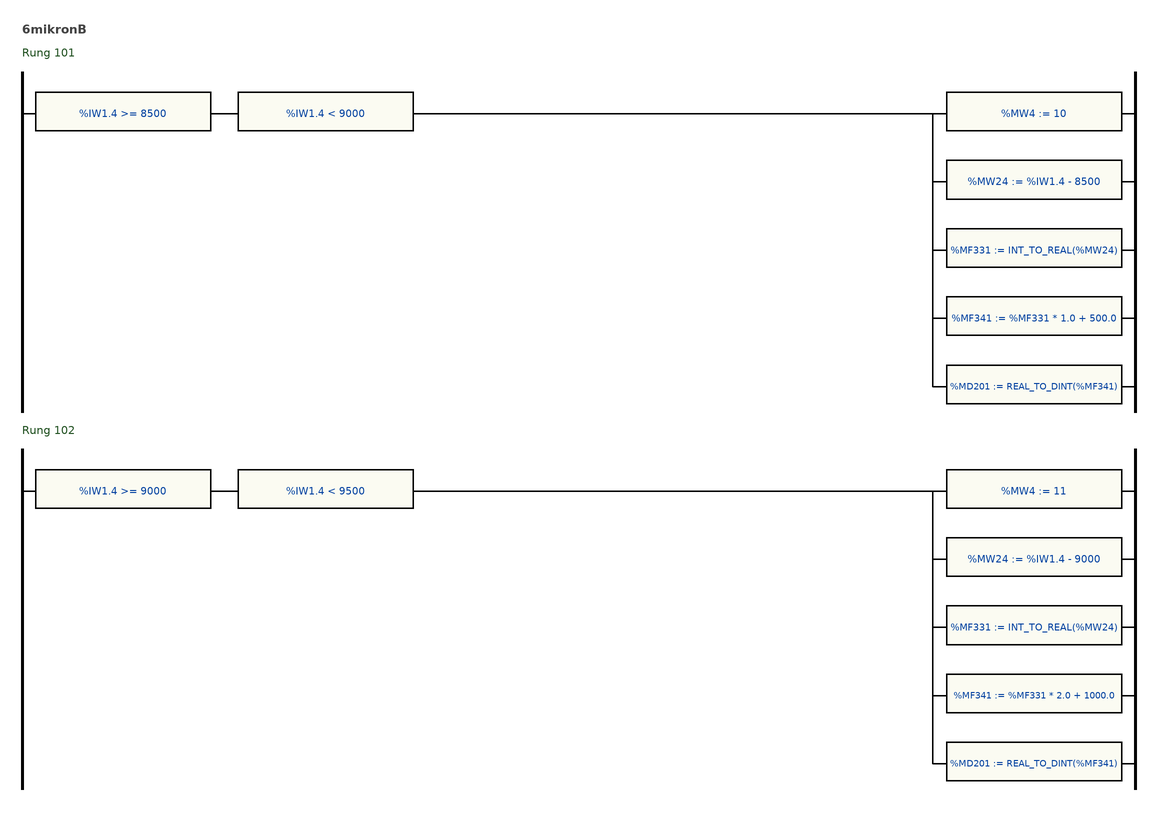
[picture p48: 6mikronB, ladder]

// Rung 101
  LD [ %IW1.4 >= 8500 ]
  AND [ %IW1.4 < 9000 ]
  [ %MW4 := 10 ]
  [ %MW24 := %IW1.4 - 8500 ]
  [ %MF331 := INT_TO_REAL ( %MW24 ) ]
  [ %MF341 := %MF331 * 1.0 + 500.0 ]
  [ %MD201 := REAL_TO_DINT ( %MF341 ) ]
  // as ST:
  //   IF %IW1.4 >= 8500 AND %IW1.4 < 9000 THEN %MW4 := 10; END_IF;
  //   IF %IW1.4 >= 8500 AND %IW1.4 < 9000 THEN %MW24 := %IW1.4 - 8500; END_IF;
  //   IF %IW1.4 >= 8500 AND %IW1.4 < 9000 THEN %MF331 := INT_TO_REAL ( %MW24 ); END_IF;
  //   IF %IW1.4 >= 8500 AND %IW1.4 < 9000 THEN %MF341 := %MF331 * 1.0 + 500.0; END_IF;
  //   IF %IW1.4 >= 8500 AND %IW1.4 < 9000 THEN %MD201 := REAL_TO_DINT ( %MF341 ); END_IF;

// Rung 102
  LD [ %IW1.4 >= 9000 ]
  AND [ %IW1.4 < 9500 ]
  [ %MW4 := 11 ]
  [ %MW24 := %IW1.4 - 9000 ]
  [ %MF331 := INT_TO_REAL ( %MW24 ) ]
  [ %MF341 := %MF331 * 2.0 + 1000.0 ]
  [ %MD201 := REAL_TO_DINT ( %MF341 ) ]
  // as ST:
  //   IF %IW1.4 >= 9000 AND %IW1.4 < 9500 THEN %MW4 := 11; END_IF;
  //   IF %IW1.4 >= 9000 AND %IW1.4 < 9500 THEN %MW24 := %IW1.4 - 9000; END_IF;
  //   IF %IW1.4 >= 9000 AND %IW1.4 < 9500 THEN %MF331 := INT_TO_REAL ( %MW24 ); END_IF;
  //   IF %IW1.4 >= 9000 AND %IW1.4 < 9500 THEN %MF341 := %MF331 * 2.0 + 1000.0; END_IF;
  //   IF %IW1.4 >= 9000 AND %IW1.4 < 9500 THEN %MD201 := REAL_TO_DINT ( %MF341 ); END_IF;

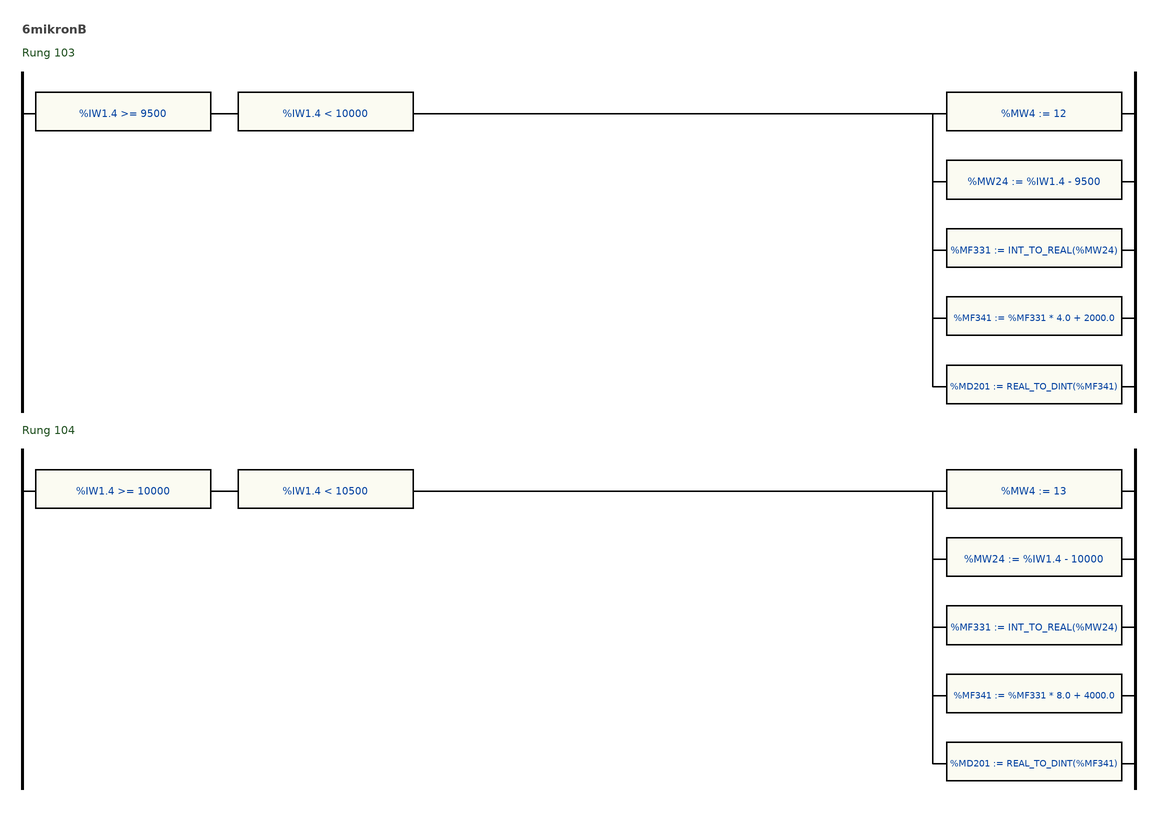

// Rung 103
  LD [ %IW1.4 >= 9500 ]
  AND [ %IW1.4 < 10000 ]
  [ %MW4 := 12 ]
  [ %MW24 := %IW1.4 - 9500 ]
  [ %MF331 := INT_TO_REAL ( %MW24 ) ]
  [ %MF341 := %MF331 * 4.0 + 2000.0 ]
  [ %MD201 := REAL_TO_DINT ( %MF341 ) ]
  // as ST:
  //   IF %IW1.4 >= 9500 AND %IW1.4 < 10000 THEN %MW4 := 12; END_IF;
  //   IF %IW1.4 >= 9500 AND %IW1.4 < 10000 THEN %MW24 := %IW1.4 - 9500; END_IF;
  //   IF %IW1.4 >= 9500 AND %IW1.4 < 10000 THEN %MF331 := INT_TO_REAL ( %MW24 ); END_IF;
  //   IF %IW1.4 >= 9500 AND %IW1.4 < 10000 THEN %MF341 := %MF331 * 4.0 + 2000.0; END_IF;
  //   IF %IW1.4 >= 9500 AND %IW1.4 < 10000 THEN %MD201 := REAL_TO_DINT ( %MF341 ); END_IF;

// Rung 104
  LD [ %IW1.4 >= 10000 ]
  AND [ %IW1.4 < 10500 ]
  [ %MW4 := 13 ]
  [ %MW24 := %IW1.4 - 10000 ]
  [ %MF331 := INT_TO_REAL ( %MW24 ) ]
  [ %MF341 := %MF331 * 8.0 + 4000.0 ]
  [ %MD201 := REAL_TO_DINT ( %MF341 ) ]
  // as ST:
  //   IF %IW1.4 >= 10000 AND %IW1.4 < 10500 THEN %MW4 := 13; END_IF;
  //   IF %IW1.4 >= 10000 AND %IW1.4 < 10500 THEN %MW24 := %IW1.4 - 10000; END_IF;
  //   IF %IW1.4 >= 10000 AND %IW1.4 < 10500 THEN %MF331 := INT_TO_REAL ( %MW24 ); END_IF;
  //   IF %IW1.4 >= 10000 AND %IW1.4 < 10500 THEN %MF341 := %MF331 * 8.0 + 4000.0; END_IF;
  //   IF %IW1.4 >= 10000 AND %IW1.4 < 10500 THEN %MD201 := REAL_TO_DINT ( %MF341 ); END_IF;

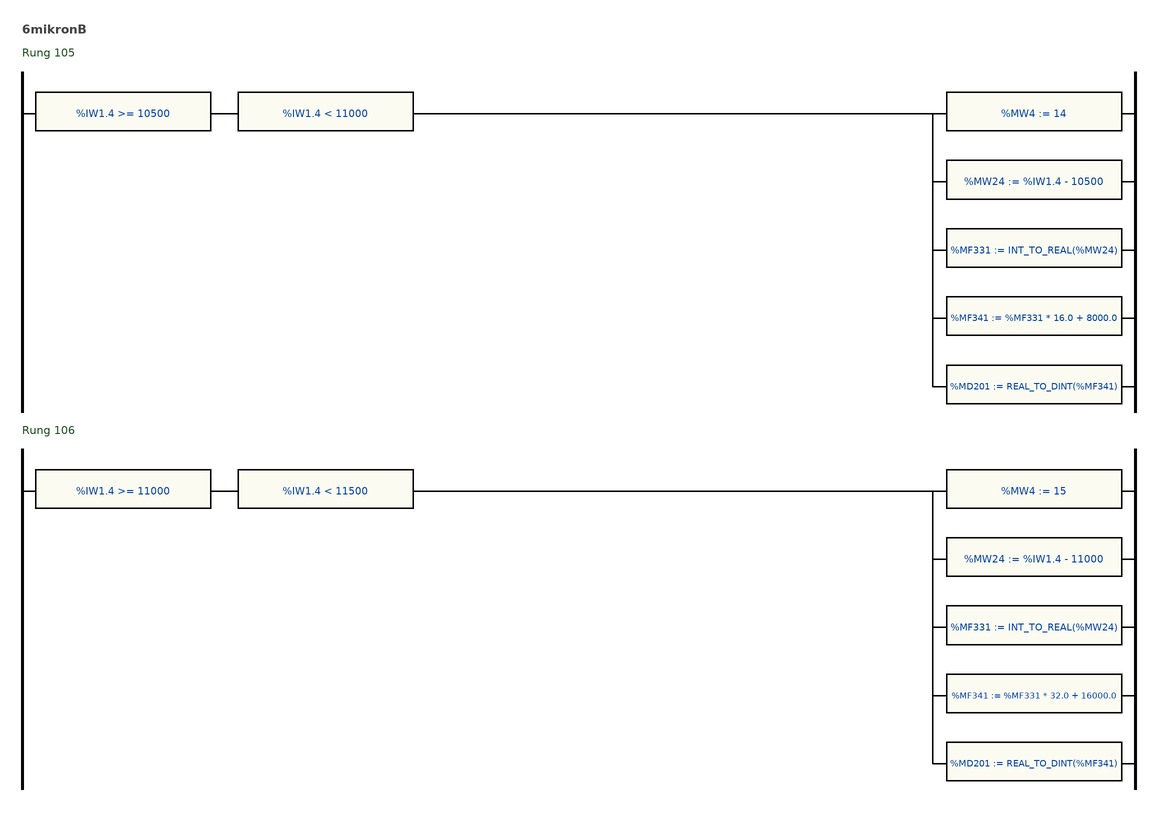

// Rung 105
  LD [ %IW1.4 >= 10500 ]
  AND [ %IW1.4 < 11000 ]
  [ %MW4 := 14 ]
  [ %MW24 := %IW1.4 - 10500 ]
  [ %MF331 := INT_TO_REAL ( %MW24 ) ]
  [ %MF341 := %MF331 * 16.0 + 8000.0 ]
  [ %MD201 := REAL_TO_DINT ( %MF341 ) ]
  // as ST:
  //   IF %IW1.4 >= 10500 AND %IW1.4 < 11000 THEN %MW4 := 14; END_IF;
  //   IF %IW1.4 >= 10500 AND %IW1.4 < 11000 THEN %MW24 := %IW1.4 - 10500; END_IF;
  //   IF %IW1.4 >= 10500 AND %IW1.4 < 11000 THEN %MF331 := INT_TO_REAL ( %MW24 ); END_IF;
  //   IF %IW1.4 >= 10500 AND %IW1.4 < 11000 THEN %MF341 := %MF331 * 16.0 + 8000.0; END_IF;
  //   IF %IW1.4 >= 10500 AND %IW1.4 < 11000 THEN %MD201 := REAL_TO_DINT ( %MF341 ); END_IF;

// Rung 106
  LD [ %IW1.4 >= 11000 ]
  AND [ %IW1.4 < 11500 ]
  [ %MW4 := 15 ]
  [ %MW24 := %IW1.4 - 11000 ]
  [ %MF331 := INT_TO_REAL ( %MW24 ) ]
  [ %MF341 := %MF331 * 32.0 + 16000.0 ]
  [ %MD201 := REAL_TO_DINT ( %MF341 ) ]
  // as ST:
  //   IF %IW1.4 >= 11000 AND %IW1.4 < 11500 THEN %MW4 := 15; END_IF;
  //   IF %IW1.4 >= 11000 AND %IW1.4 < 11500 THEN %MW24 := %IW1.4 - 11000; END_IF;
  //   IF %IW1.4 >= 11000 AND %IW1.4 < 11500 THEN %MF331 := INT_TO_REAL ( %MW24 ); END_IF;
  //   IF %IW1.4 >= 11000 AND %IW1.4 < 11500 THEN %MF341 := %MF331 * 32.0 + 16000.0; END_IF;
  //   IF %IW1.4 >= 11000 AND %IW1.4 < 11500 THEN %MD201 := REAL_TO_DINT ( %MF341 ); END_IF;

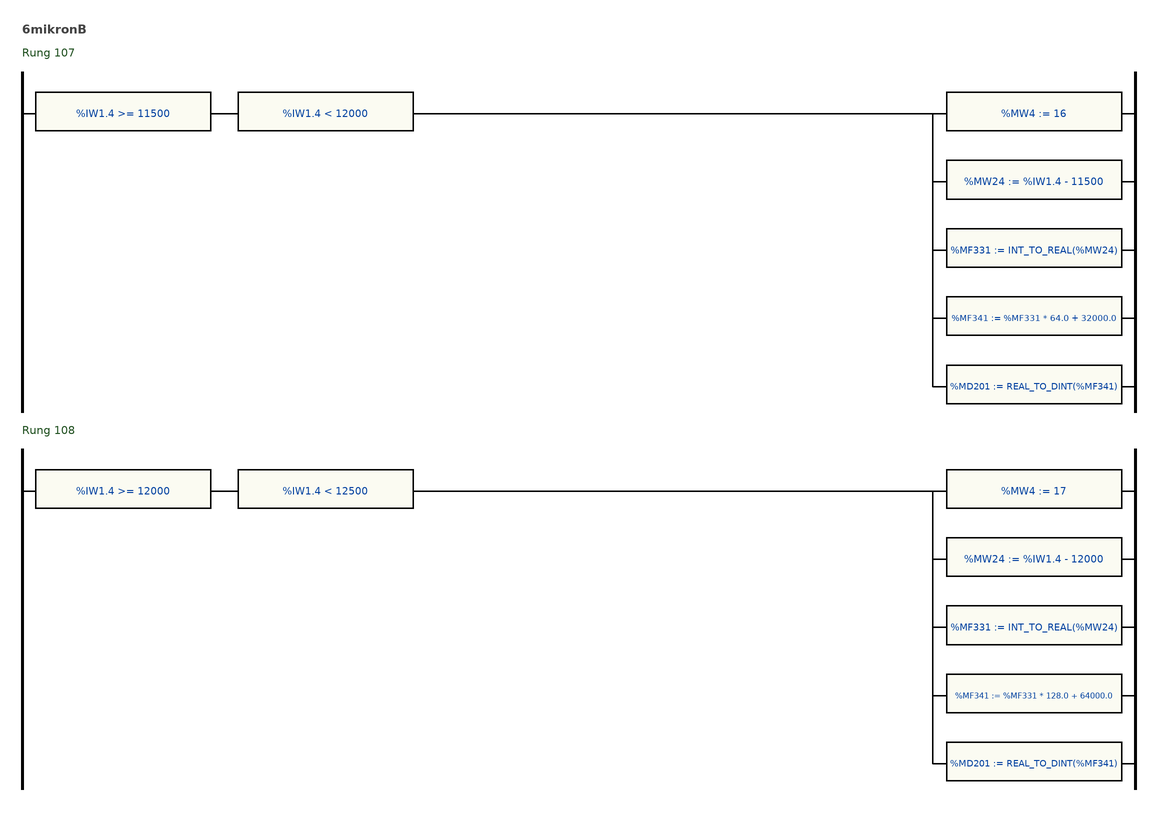

// Rung 107
  LD [ %IW1.4 >= 11500 ]
  AND [ %IW1.4 < 12000 ]
  [ %MW4 := 16 ]
  [ %MW24 := %IW1.4 - 11500 ]
  [ %MF331 := INT_TO_REAL ( %MW24 ) ]
  [ %MF341 := %MF331 * 64.0 + 32000.0 ]
  [ %MD201 := REAL_TO_DINT ( %MF341 ) ]
  // as ST:
  //   IF %IW1.4 >= 11500 AND %IW1.4 < 12000 THEN %MW4 := 16; END_IF;
  //   IF %IW1.4 >= 11500 AND %IW1.4 < 12000 THEN %MW24 := %IW1.4 - 11500; END_IF;
  //   IF %IW1.4 >= 11500 AND %IW1.4 < 12000 THEN %MF331 := INT_TO_REAL ( %MW24 ); END_IF;
  //   IF %IW1.4 >= 11500 AND %IW1.4 < 12000 THEN %MF341 := %MF331 * 64.0 + 32000.0; END_IF;
  //   IF %IW1.4 >= 11500 AND %IW1.4 < 12000 THEN %MD201 := REAL_TO_DINT ( %MF341 ); END_IF;

// Rung 108
  LD [ %IW1.4 >= 12000 ]
  AND [ %IW1.4 < 12500 ]
  [ %MW4 := 17 ]
  [ %MW24 := %IW1.4 - 12000 ]
  [ %MF331 := INT_TO_REAL ( %MW24 ) ]
  [ %MF341 := %MF331 * 128.0 + 64000.0 ]
  [ %MD201 := REAL_TO_DINT ( %MF341 ) ]
  // as ST:
  //   IF %IW1.4 >= 12000 AND %IW1.4 < 12500 THEN %MW4 := 17; END_IF;
  //   IF %IW1.4 >= 12000 AND %IW1.4 < 12500 THEN %MW24 := %IW1.4 - 12000; END_IF;
  //   IF %IW1.4 >= 12000 AND %IW1.4 < 12500 THEN %MF331 := INT_TO_REAL ( %MW24 ); END_IF;
  //   IF %IW1.4 >= 12000 AND %IW1.4 < 12500 THEN %MF341 := %MF331 * 128.0 + 64000.0; END_IF;
  //   IF %IW1.4 >= 12000 AND %IW1.4 < 12500 THEN %MD201 := REAL_TO_DINT ( %MF341 ); END_IF;

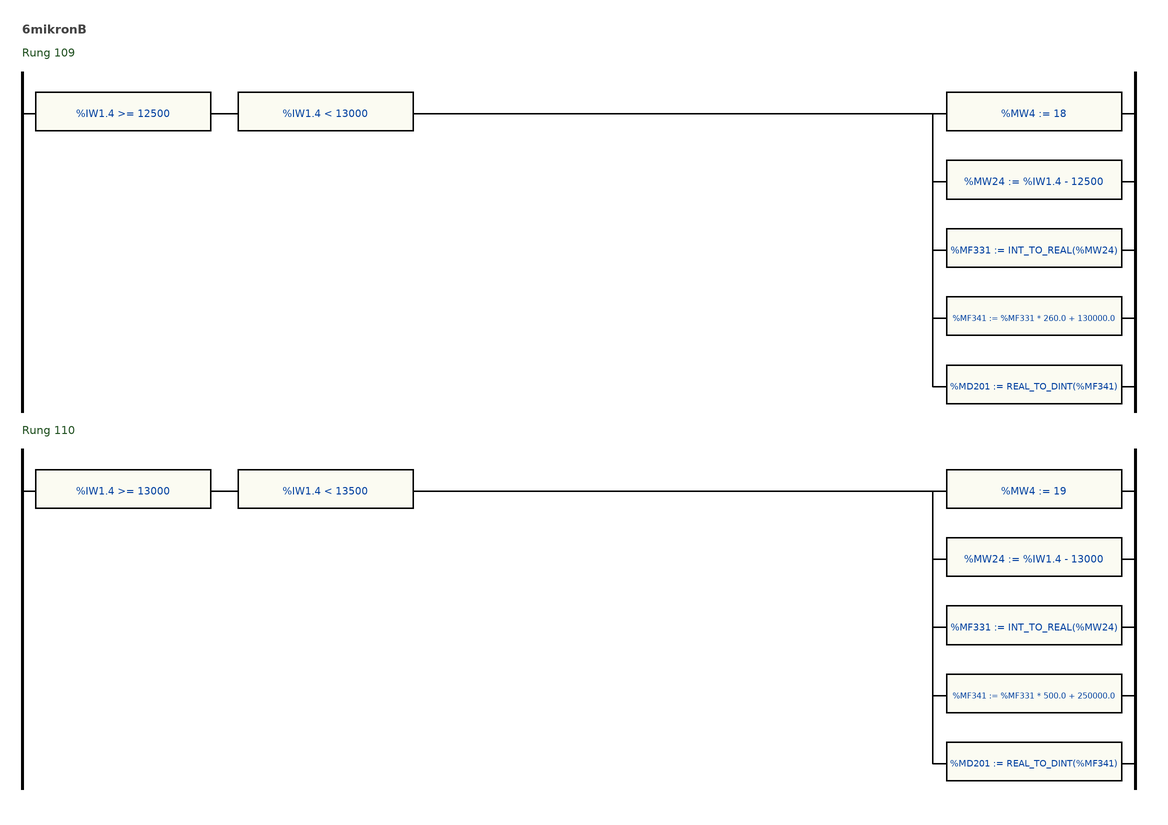

// Rung 109
  LD [ %IW1.4 >= 12500 ]
  AND [ %IW1.4 < 13000 ]
  [ %MW4 := 18 ]
  [ %MW24 := %IW1.4 - 12500 ]
  [ %MF331 := INT_TO_REAL ( %MW24 ) ]
  [ %MF341 := %MF331 * 260.0 + 130000.0 ]
  [ %MD201 := REAL_TO_DINT ( %MF341 ) ]
  // as ST:
  //   IF %IW1.4 >= 12500 AND %IW1.4 < 13000 THEN %MW4 := 18; END_IF;
  //   IF %IW1.4 >= 12500 AND %IW1.4 < 13000 THEN %MW24 := %IW1.4 - 12500; END_IF;
  //   IF %IW1.4 >= 12500 AND %IW1.4 < 13000 THEN %MF331 := INT_TO_REAL ( %MW24 ); END_IF;
  //   IF %IW1.4 >= 12500 AND %IW1.4 < 13000 THEN %MF341 := %MF331 * 260.0 + 130000.0; END_IF;
  //   IF %IW1.4 >= 12500 AND %IW1.4 < 13000 THEN %MD201 := REAL_TO_DINT ( %MF341 ); END_IF;

// Rung 110
  LD [ %IW1.4 >= 13000 ]
  AND [ %IW1.4 < 13500 ]
  [ %MW4 := 19 ]
  [ %MW24 := %IW1.4 - 13000 ]
  [ %MF331 := INT_TO_REAL ( %MW24 ) ]
  [ %MF341 := %MF331 * 500.0 + 250000.0 ]
  [ %MD201 := REAL_TO_DINT ( %MF341 ) ]
  // as ST:
  //   IF %IW1.4 >= 13000 AND %IW1.4 < 13500 THEN %MW4 := 19; END_IF;
  //   IF %IW1.4 >= 13000 AND %IW1.4 < 13500 THEN %MW24 := %IW1.4 - 13000; END_IF;
  //   IF %IW1.4 >= 13000 AND %IW1.4 < 13500 THEN %MF331 := INT_TO_REAL ( %MW24 ); END_IF;
  //   IF %IW1.4 >= 13000 AND %IW1.4 < 13500 THEN %MF341 := %MF331 * 500.0 + 250000.0; END_IF;
  //   IF %IW1.4 >= 13000 AND %IW1.4 < 13500 THEN %MD201 := REAL_TO_DINT ( %MF341 ); END_IF;

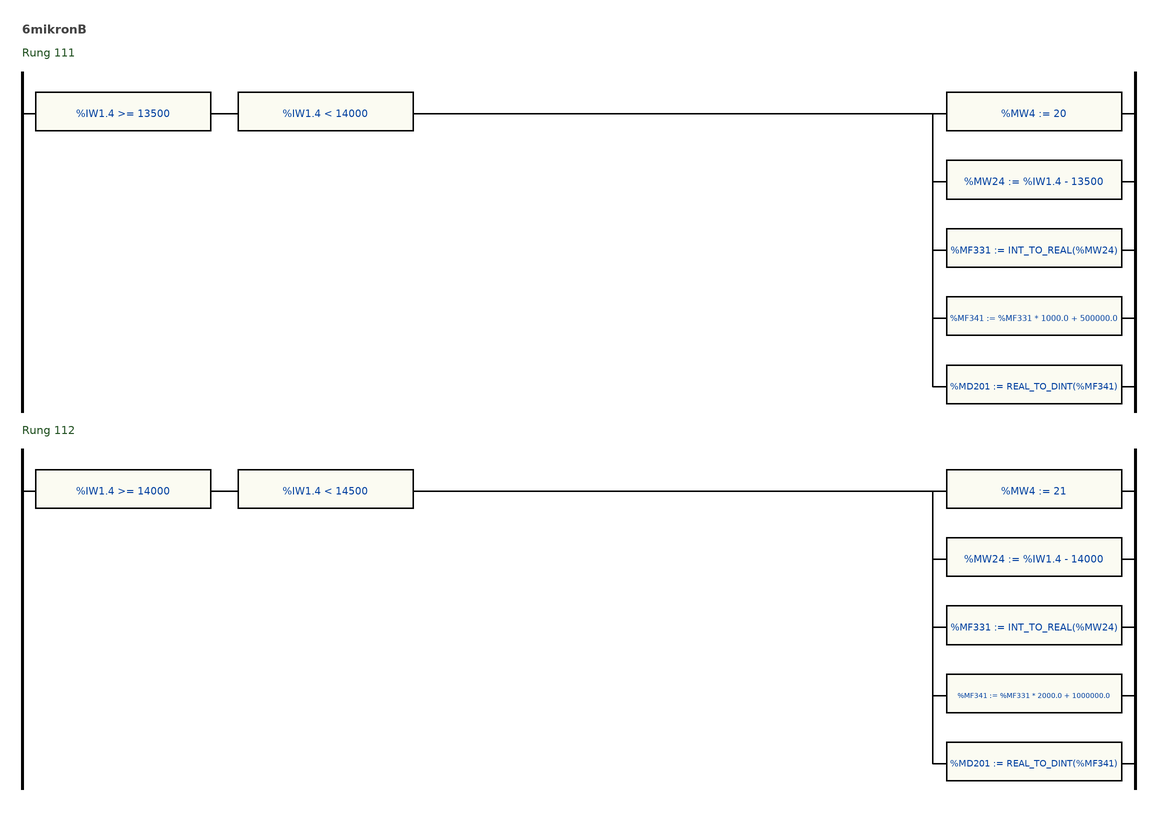

// Rung 111
  LD [ %IW1.4 >= 13500 ]
  AND [ %IW1.4 < 14000 ]
  [ %MW4 := 20 ]
  [ %MW24 := %IW1.4 - 13500 ]
  [ %MF331 := INT_TO_REAL ( %MW24 ) ]
  [ %MF341 := %MF331 * 1000.0 + 500000.0 ]
  [ %MD201 := REAL_TO_DINT ( %MF341 ) ]
  // as ST:
  //   IF %IW1.4 >= 13500 AND %IW1.4 < 14000 THEN %MW4 := 20; END_IF;
  //   IF %IW1.4 >= 13500 AND %IW1.4 < 14000 THEN %MW24 := %IW1.4 - 13500; END_IF;
  //   IF %IW1.4 >= 13500 AND %IW1.4 < 14000 THEN %MF331 := INT_TO_REAL ( %MW24 ); END_IF;
  //   IF %IW1.4 >= 13500 AND %IW1.4 < 14000 THEN %MF341 := %MF331 * 1000.0 + 500000.0; END_IF;
  //   IF %IW1.4 >= 13500 AND %IW1.4 < 14000 THEN %MD201 := REAL_TO_DINT ( %MF341 ); END_IF;

// Rung 112
  LD [ %IW1.4 >= 14000 ]
  AND [ %IW1.4 < 14500 ]
  [ %MW4 := 21 ]
  [ %MW24 := %IW1.4 - 14000 ]
  [ %MF331 := INT_TO_REAL ( %MW24 ) ]
  [ %MF341 := %MF331 * 2000.0 + 1000000.0 ]
  [ %MD201 := REAL_TO_DINT ( %MF341 ) ]
  // as ST:
  //   IF %IW1.4 >= 14000 AND %IW1.4 < 14500 THEN %MW4 := 21; END_IF;
  //   IF %IW1.4 >= 14000 AND %IW1.4 < 14500 THEN %MW24 := %IW1.4 - 14000; END_IF;
  //   IF %IW1.4 >= 14000 AND %IW1.4 < 14500 THEN %MF331 := INT_TO_REAL ( %MW24 ); END_IF;
  //   IF %IW1.4 >= 14000 AND %IW1.4 < 14500 THEN %MF341 := %MF331 * 2000.0 + 1000000.0; END_IF;
  //   IF %IW1.4 >= 14000 AND %IW1.4 < 14500 THEN %MD201 := REAL_TO_DINT ( %MF341 ); END_IF;

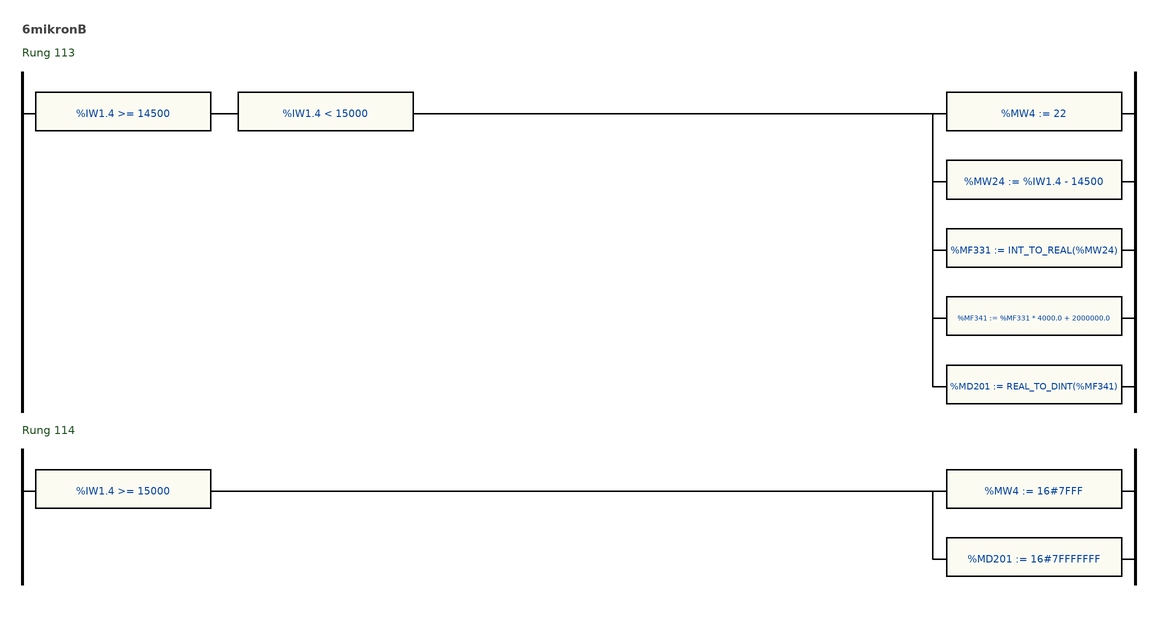

// Rung 113
  LD [ %IW1.4 >= 14500 ]
  AND [ %IW1.4 < 15000 ]
  [ %MW4 := 22 ]
  [ %MW24 := %IW1.4 - 14500 ]
  [ %MF331 := INT_TO_REAL ( %MW24 ) ]
  [ %MF341 := %MF331 * 4000.0 + 2000000.0 ]
  [ %MD201 := REAL_TO_DINT ( %MF341 ) ]
  // as ST:
  //   IF %IW1.4 >= 14500 AND %IW1.4 < 15000 THEN %MW4 := 22; END_IF;
  //   IF %IW1.4 >= 14500 AND %IW1.4 < 15000 THEN %MW24 := %IW1.4 - 14500; END_IF;
  //   IF %IW1.4 >= 14500 AND %IW1.4 < 15000 THEN %MF331 := INT_TO_REAL ( %MW24 ); END_IF;
  //   IF %IW1.4 >= 14500 AND %IW1.4 < 15000 THEN %MF341 := %MF331 * 4000.0 + 2000000.0; END_IF;
  //   IF %IW1.4 >= 14500 AND %IW1.4 < 15000 THEN %MD201 := REAL_TO_DINT ( %MF341 ); END_IF;

// Rung 114
  LD [ %IW1.4 >= 15000 ]
  [ %MW4 := 16#7FFF ]
  [ %MD201 := 16#7FFFFFFF ]
  // as ST:
  //   IF %IW1.4 >= 15000 THEN %MW4 := 16#7FFF; END_IF;
  //   IF %IW1.4 >= 15000 THEN %MD201 := 16#7FFFFFFF; END_IF;

POU 14mikronB
  (* SectionNumber=6 *)

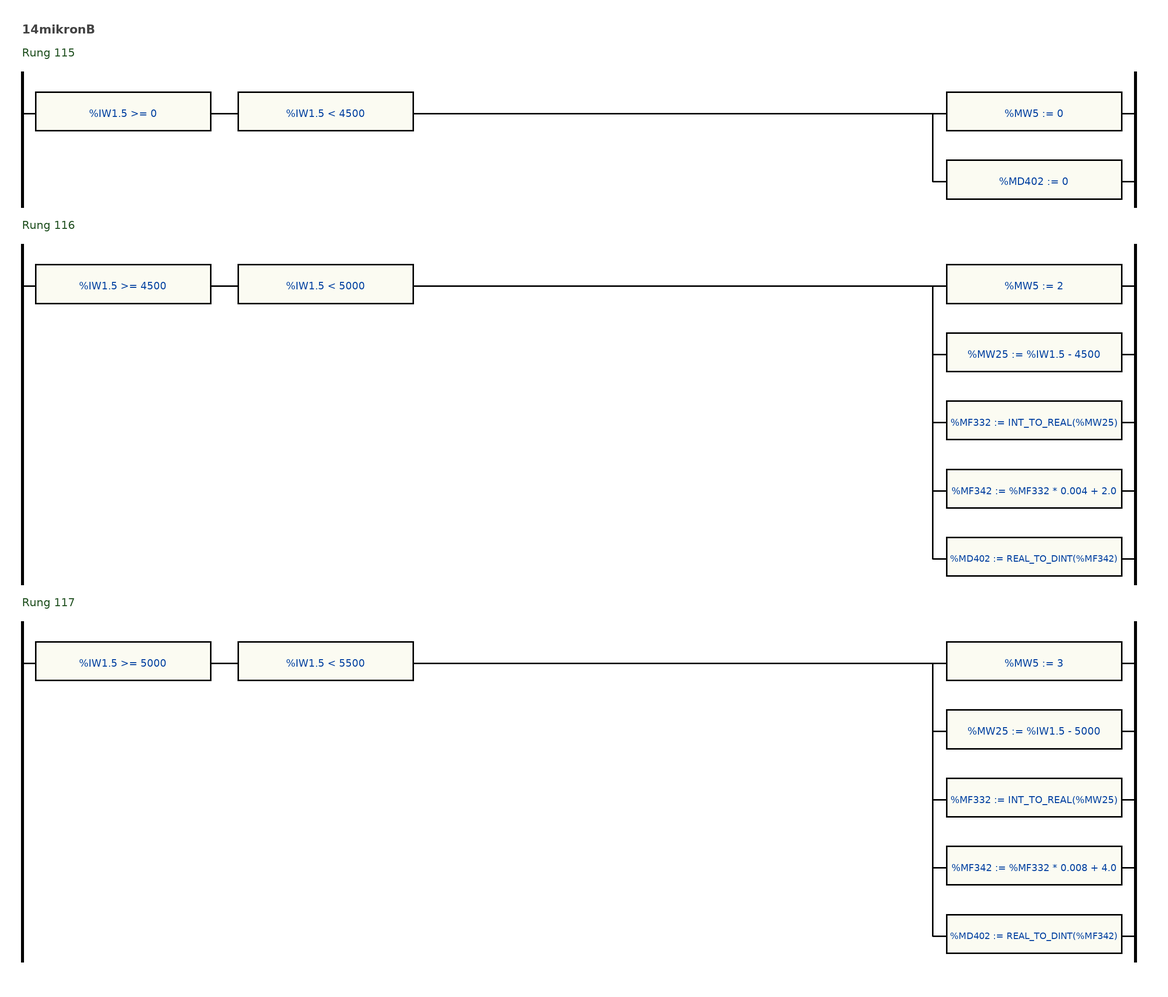

// Rung 115
  LD [ %IW1.5 >= 0 ]
  AND [ %IW1.5 < 4500 ]
  [ %MW5 := 0 ]
  [ %MD402 := 0 ]
  // as ST:
  //   IF %IW1.5 >= 0 AND %IW1.5 < 4500 THEN %MW5 := 0; END_IF;
  //   IF %IW1.5 >= 0 AND %IW1.5 < 4500 THEN %MD402 := 0; END_IF;

// Rung 116
  LD [ %IW1.5 >= 4500 ]
  AND [ %IW1.5 < 5000 ]
  [ %MW5 := 2 ]
  [ %MW25 := %IW1.5 - 4500 ]
  [ %MF332 := INT_TO_REAL ( %MW25 ) ]
  [ %MF342 := %MF332 * 0.004 + 2.0 ]
  [ %MD402 := REAL_TO_DINT ( %MF342 ) ]
  // as ST:
  //   IF %IW1.5 >= 4500 AND %IW1.5 < 5000 THEN %MW5 := 2; END_IF;
  //   IF %IW1.5 >= 4500 AND %IW1.5 < 5000 THEN %MW25 := %IW1.5 - 4500; END_IF;
  //   IF %IW1.5 >= 4500 AND %IW1.5 < 5000 THEN %MF332 := INT_TO_REAL ( %MW25 ); END_IF;
  //   IF %IW1.5 >= 4500 AND %IW1.5 < 5000 THEN %MF342 := %MF332 * 0.004 + 2.0; END_IF;
  //   IF %IW1.5 >= 4500 AND %IW1.5 < 5000 THEN %MD402 := REAL_TO_DINT ( %MF342 ); END_IF;

// Rung 117
  LD [ %IW1.5 >= 5000 ]
  AND [ %IW1.5 < 5500 ]
  [ %MW5 := 3 ]
  [ %MW25 := %IW1.5 - 5000 ]
  [ %MF332 := INT_TO_REAL ( %MW25 ) ]
  [ %MF342 := %MF332 * 0.008 + 4.0 ]
  [ %MD402 := REAL_TO_DINT ( %MF342 ) ]
  // as ST:
  //   IF %IW1.5 >= 5000 AND %IW1.5 < 5500 THEN %MW5 := 3; END_IF;
  //   IF %IW1.5 >= 5000 AND %IW1.5 < 5500 THEN %MW25 := %IW1.5 - 5000; END_IF;
  //   IF %IW1.5 >= 5000 AND %IW1.5 < 5500 THEN %MF332 := INT_TO_REAL ( %MW25 ); END_IF;
  //   IF %IW1.5 >= 5000 AND %IW1.5 < 5500 THEN %MF342 := %MF332 * 0.008 + 4.0; END_IF;
  //   IF %IW1.5 >= 5000 AND %IW1.5 < 5500 THEN %MD402 := REAL_TO_DINT ( %MF342 ); END_IF;

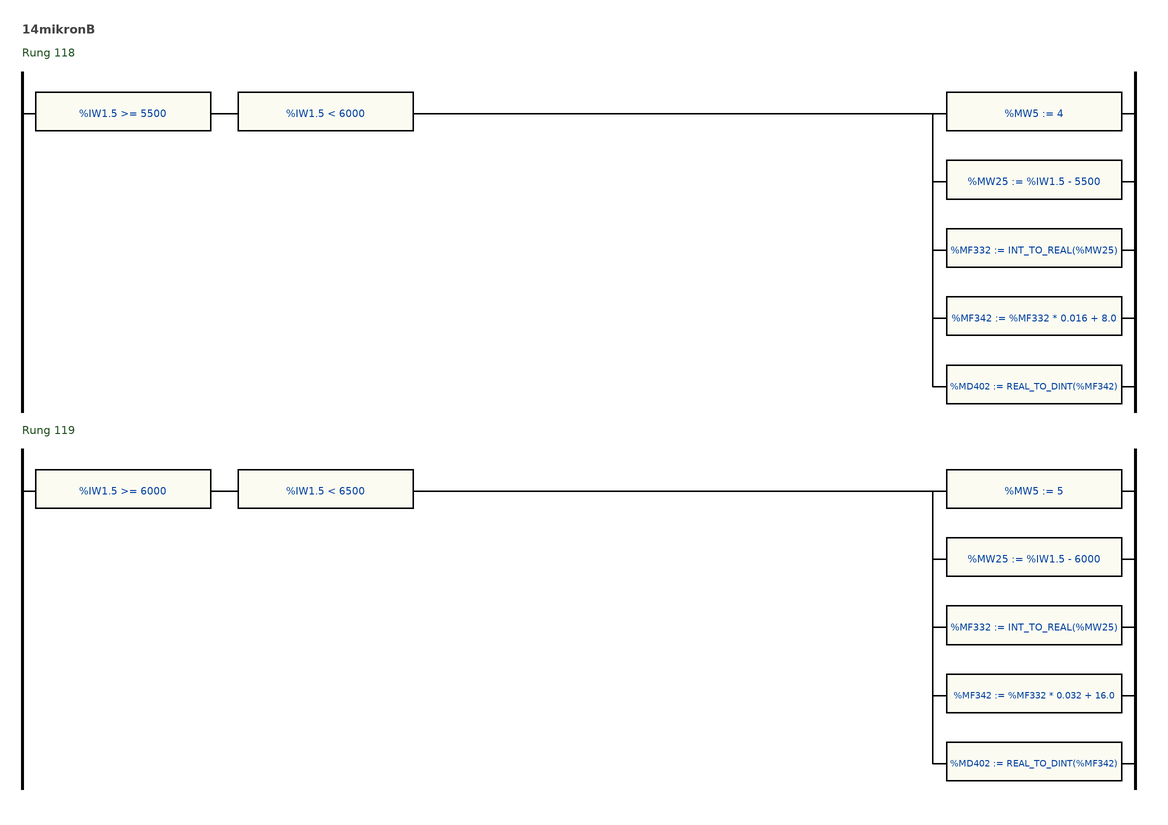

// Rung 118
  LD [ %IW1.5 >= 5500 ]
  AND [ %IW1.5 < 6000 ]
  [ %MW5 := 4 ]
  [ %MW25 := %IW1.5 - 5500 ]
  [ %MF332 := INT_TO_REAL ( %MW25 ) ]
  [ %MF342 := %MF332 * 0.016 + 8.0 ]
  [ %MD402 := REAL_TO_DINT ( %MF342 ) ]
  // as ST:
  //   IF %IW1.5 >= 5500 AND %IW1.5 < 6000 THEN %MW5 := 4; END_IF;
  //   IF %IW1.5 >= 5500 AND %IW1.5 < 6000 THEN %MW25 := %IW1.5 - 5500; END_IF;
  //   IF %IW1.5 >= 5500 AND %IW1.5 < 6000 THEN %MF332 := INT_TO_REAL ( %MW25 ); END_IF;
  //   IF %IW1.5 >= 5500 AND %IW1.5 < 6000 THEN %MF342 := %MF332 * 0.016 + 8.0; END_IF;
  //   IF %IW1.5 >= 5500 AND %IW1.5 < 6000 THEN %MD402 := REAL_TO_DINT ( %MF342 ); END_IF;

// Rung 119
  LD [ %IW1.5 >= 6000 ]
  AND [ %IW1.5 < 6500 ]
  [ %MW5 := 5 ]
  [ %MW25 := %IW1.5 - 6000 ]
  [ %MF332 := INT_TO_REAL ( %MW25 ) ]
  [ %MF342 := %MF332 * 0.032 + 16.0 ]
  [ %MD402 := REAL_TO_DINT ( %MF342 ) ]
  // as ST:
  //   IF %IW1.5 >= 6000 AND %IW1.5 < 6500 THEN %MW5 := 5; END_IF;
  //   IF %IW1.5 >= 6000 AND %IW1.5 < 6500 THEN %MW25 := %IW1.5 - 6000; END_IF;
  //   IF %IW1.5 >= 6000 AND %IW1.5 < 6500 THEN %MF332 := INT_TO_REAL ( %MW25 ); END_IF;
  //   IF %IW1.5 >= 6000 AND %IW1.5 < 6500 THEN %MF342 := %MF332 * 0.032 + 16.0; END_IF;
  //   IF %IW1.5 >= 6000 AND %IW1.5 < 6500 THEN %MD402 := REAL_TO_DINT ( %MF342 ); END_IF;

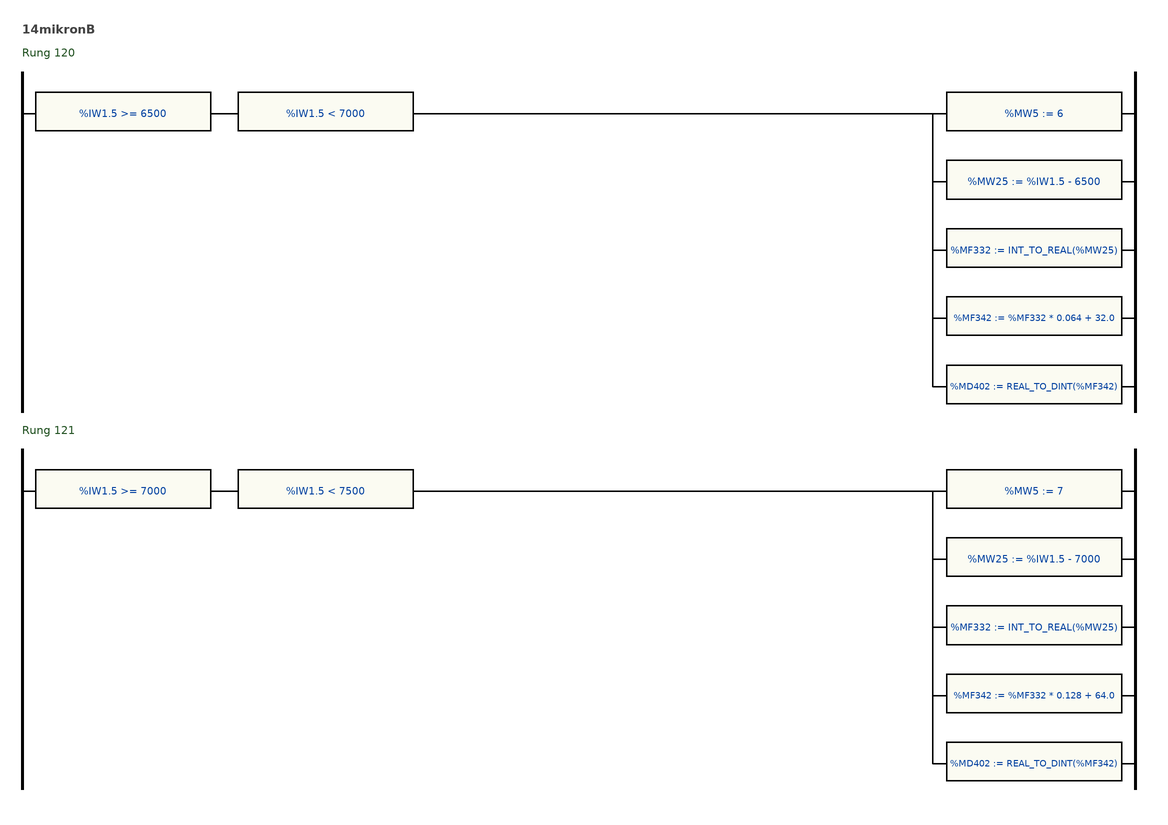

// Rung 120
  LD [ %IW1.5 >= 6500 ]
  AND [ %IW1.5 < 7000 ]
  [ %MW5 := 6 ]
  [ %MW25 := %IW1.5 - 6500 ]
  [ %MF332 := INT_TO_REAL ( %MW25 ) ]
  [ %MF342 := %MF332 * 0.064 + 32.0 ]
  [ %MD402 := REAL_TO_DINT ( %MF342 ) ]
  // as ST:
  //   IF %IW1.5 >= 6500 AND %IW1.5 < 7000 THEN %MW5 := 6; END_IF;
  //   IF %IW1.5 >= 6500 AND %IW1.5 < 7000 THEN %MW25 := %IW1.5 - 6500; END_IF;
  //   IF %IW1.5 >= 6500 AND %IW1.5 < 7000 THEN %MF332 := INT_TO_REAL ( %MW25 ); END_IF;
  //   IF %IW1.5 >= 6500 AND %IW1.5 < 7000 THEN %MF342 := %MF332 * 0.064 + 32.0; END_IF;
  //   IF %IW1.5 >= 6500 AND %IW1.5 < 7000 THEN %MD402 := REAL_TO_DINT ( %MF342 ); END_IF;

// Rung 121
  LD [ %IW1.5 >= 7000 ]
  AND [ %IW1.5 < 7500 ]
  [ %MW5 := 7 ]
  [ %MW25 := %IW1.5 - 7000 ]
  [ %MF332 := INT_TO_REAL ( %MW25 ) ]
  [ %MF342 := %MF332 * 0.128 + 64.0 ]
  [ %MD402 := REAL_TO_DINT ( %MF342 ) ]
  // as ST:
  //   IF %IW1.5 >= 7000 AND %IW1.5 < 7500 THEN %MW5 := 7; END_IF;
  //   IF %IW1.5 >= 7000 AND %IW1.5 < 7500 THEN %MW25 := %IW1.5 - 7000; END_IF;
  //   IF %IW1.5 >= 7000 AND %IW1.5 < 7500 THEN %MF332 := INT_TO_REAL ( %MW25 ); END_IF;
  //   IF %IW1.5 >= 7000 AND %IW1.5 < 7500 THEN %MF342 := %MF332 * 0.128 + 64.0; END_IF;
  //   IF %IW1.5 >= 7000 AND %IW1.5 < 7500 THEN %MD402 := REAL_TO_DINT ( %MF342 ); END_IF;

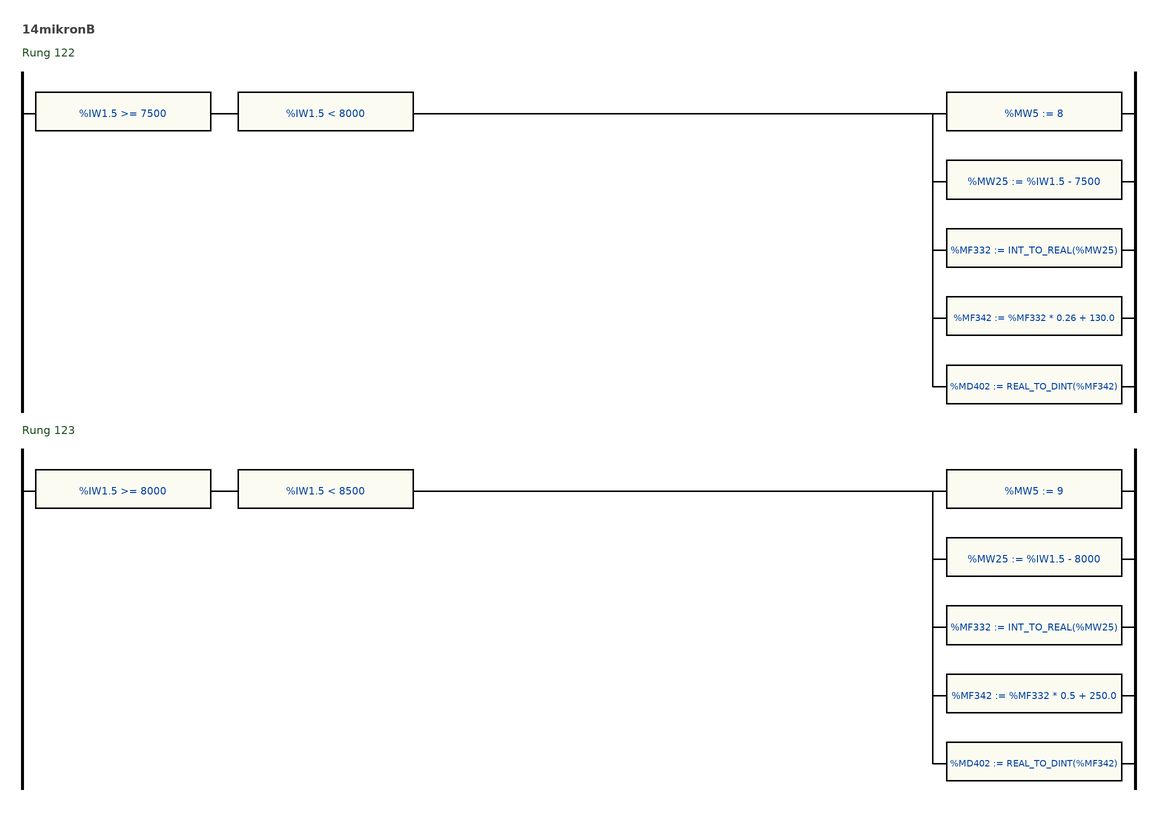

// Rung 122
  LD [ %IW1.5 >= 7500 ]
  AND [ %IW1.5 < 8000 ]
  [ %MW5 := 8 ]
  [ %MW25 := %IW1.5 - 7500 ]
  [ %MF332 := INT_TO_REAL ( %MW25 ) ]
  [ %MF342 := %MF332 * 0.26 + 130.0 ]
  [ %MD402 := REAL_TO_DINT ( %MF342 ) ]
  // as ST:
  //   IF %IW1.5 >= 7500 AND %IW1.5 < 8000 THEN %MW5 := 8; END_IF;
  //   IF %IW1.5 >= 7500 AND %IW1.5 < 8000 THEN %MW25 := %IW1.5 - 7500; END_IF;
  //   IF %IW1.5 >= 7500 AND %IW1.5 < 8000 THEN %MF332 := INT_TO_REAL ( %MW25 ); END_IF;
  //   IF %IW1.5 >= 7500 AND %IW1.5 < 8000 THEN %MF342 := %MF332 * 0.26 + 130.0; END_IF;
  //   IF %IW1.5 >= 7500 AND %IW1.5 < 8000 THEN %MD402 := REAL_TO_DINT ( %MF342 ); END_IF;

// Rung 123
  LD [ %IW1.5 >= 8000 ]
  AND [ %IW1.5 < 8500 ]
  [ %MW5 := 9 ]
  [ %MW25 := %IW1.5 - 8000 ]
  [ %MF332 := INT_TO_REAL ( %MW25 ) ]
  [ %MF342 := %MF332 * 0.5 + 250.0 ]
  [ %MD402 := REAL_TO_DINT ( %MF342 ) ]
  // as ST:
  //   IF %IW1.5 >= 8000 AND %IW1.5 < 8500 THEN %MW5 := 9; END_IF;
  //   IF %IW1.5 >= 8000 AND %IW1.5 < 8500 THEN %MW25 := %IW1.5 - 8000; END_IF;
  //   IF %IW1.5 >= 8000 AND %IW1.5 < 8500 THEN %MF332 := INT_TO_REAL ( %MW25 ); END_IF;
  //   IF %IW1.5 >= 8000 AND %IW1.5 < 8500 THEN %MF342 := %MF332 * 0.5 + 250.0; END_IF;
  //   IF %IW1.5 >= 8000 AND %IW1.5 < 8500 THEN %MD402 := REAL_TO_DINT ( %MF342 ); END_IF;

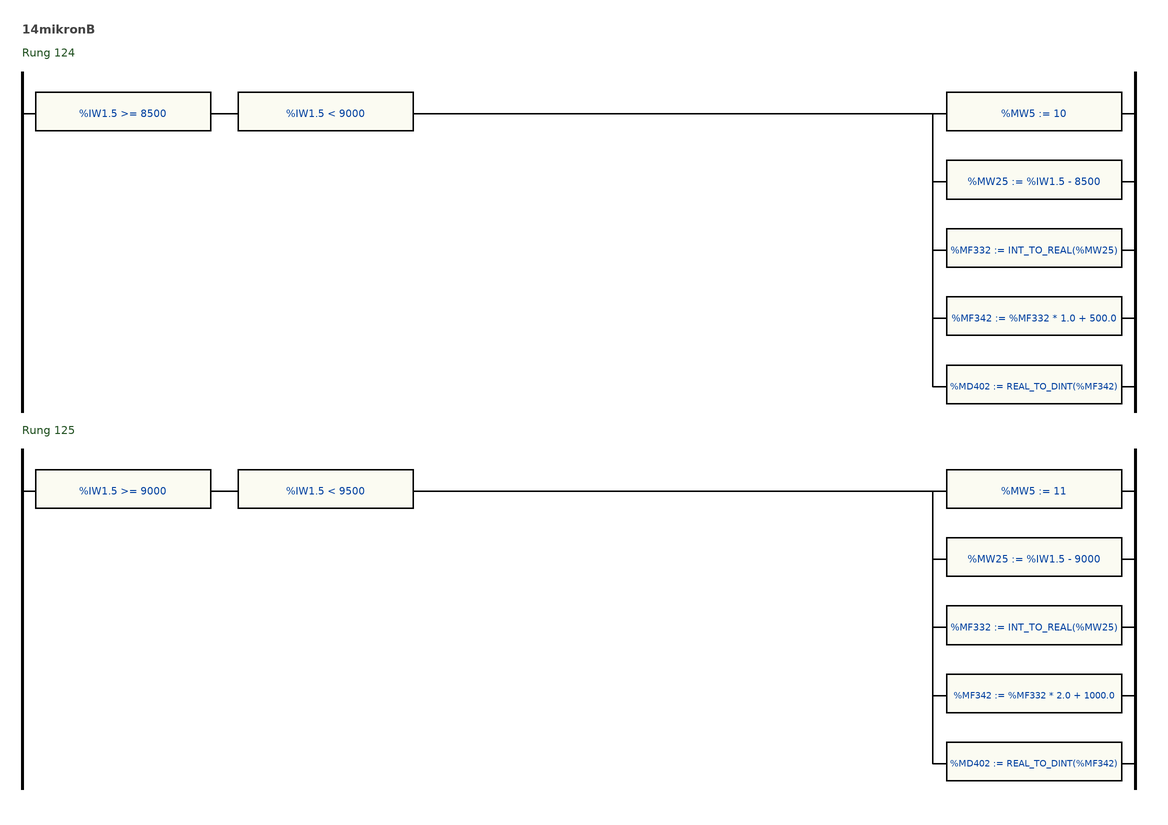

// Rung 124
  LD [ %IW1.5 >= 8500 ]
  AND [ %IW1.5 < 9000 ]
  [ %MW5 := 10 ]
  [ %MW25 := %IW1.5 - 8500 ]
  [ %MF332 := INT_TO_REAL ( %MW25 ) ]
  [ %MF342 := %MF332 * 1.0 + 500.0 ]
  [ %MD402 := REAL_TO_DINT ( %MF342 ) ]
  // as ST:
  //   IF %IW1.5 >= 8500 AND %IW1.5 < 9000 THEN %MW5 := 10; END_IF;
  //   IF %IW1.5 >= 8500 AND %IW1.5 < 9000 THEN %MW25 := %IW1.5 - 8500; END_IF;
  //   IF %IW1.5 >= 8500 AND %IW1.5 < 9000 THEN %MF332 := INT_TO_REAL ( %MW25 ); END_IF;
  //   IF %IW1.5 >= 8500 AND %IW1.5 < 9000 THEN %MF342 := %MF332 * 1.0 + 500.0; END_IF;
  //   IF %IW1.5 >= 8500 AND %IW1.5 < 9000 THEN %MD402 := REAL_TO_DINT ( %MF342 ); END_IF;

// Rung 125
  LD [ %IW1.5 >= 9000 ]
  AND [ %IW1.5 < 9500 ]
  [ %MW5 := 11 ]
  [ %MW25 := %IW1.5 - 9000 ]
  [ %MF332 := INT_TO_REAL ( %MW25 ) ]
  [ %MF342 := %MF332 * 2.0 + 1000.0 ]
  [ %MD402 := REAL_TO_DINT ( %MF342 ) ]
  // as ST:
  //   IF %IW1.5 >= 9000 AND %IW1.5 < 9500 THEN %MW5 := 11; END_IF;
  //   IF %IW1.5 >= 9000 AND %IW1.5 < 9500 THEN %MW25 := %IW1.5 - 9000; END_IF;
  //   IF %IW1.5 >= 9000 AND %IW1.5 < 9500 THEN %MF332 := INT_TO_REAL ( %MW25 ); END_IF;
  //   IF %IW1.5 >= 9000 AND %IW1.5 < 9500 THEN %MF342 := %MF332 * 2.0 + 1000.0; END_IF;
  //   IF %IW1.5 >= 9000 AND %IW1.5 < 9500 THEN %MD402 := REAL_TO_DINT ( %MF342 ); END_IF;

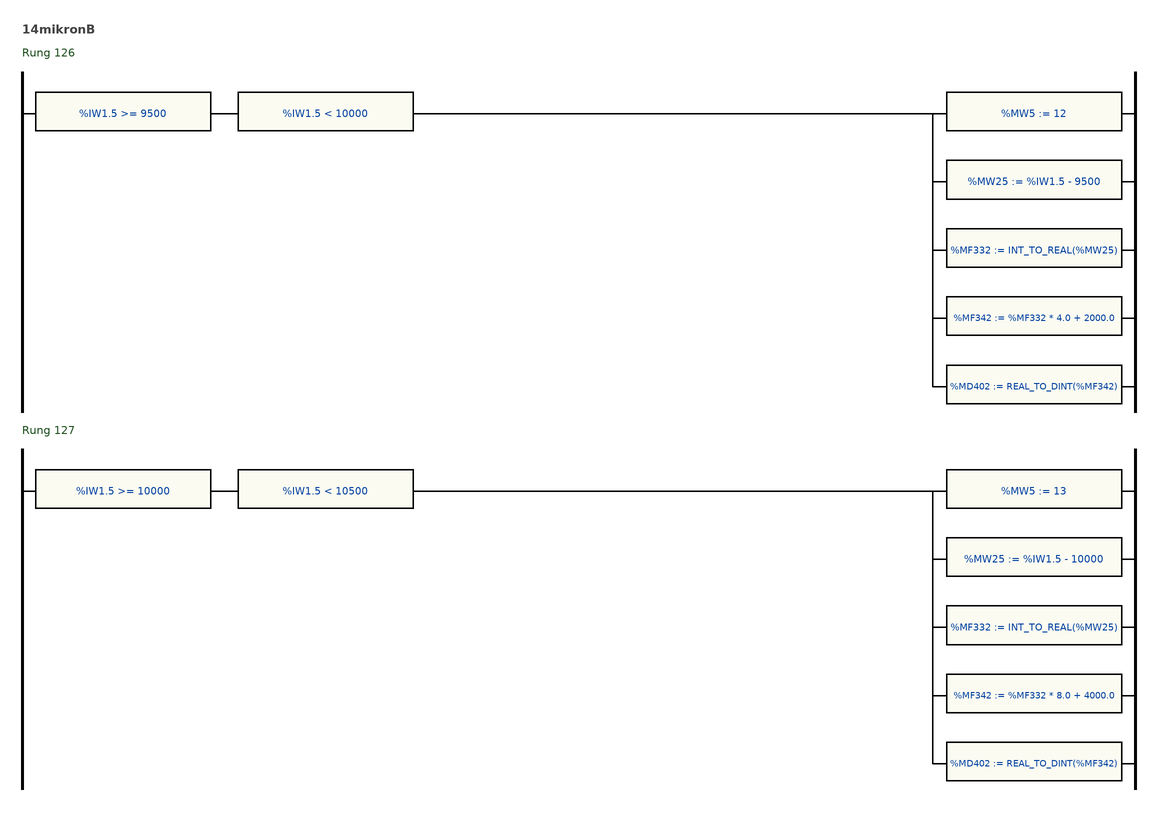

// Rung 126
  LD [ %IW1.5 >= 9500 ]
  AND [ %IW1.5 < 10000 ]
  [ %MW5 := 12 ]
  [ %MW25 := %IW1.5 - 9500 ]
  [ %MF332 := INT_TO_REAL ( %MW25 ) ]
  [ %MF342 := %MF332 * 4.0 + 2000.0 ]
  [ %MD402 := REAL_TO_DINT ( %MF342 ) ]
  // as ST:
  //   IF %IW1.5 >= 9500 AND %IW1.5 < 10000 THEN %MW5 := 12; END_IF;
  //   IF %IW1.5 >= 9500 AND %IW1.5 < 10000 THEN %MW25 := %IW1.5 - 9500; END_IF;
  //   IF %IW1.5 >= 9500 AND %IW1.5 < 10000 THEN %MF332 := INT_TO_REAL ( %MW25 ); END_IF;
  //   IF %IW1.5 >= 9500 AND %IW1.5 < 10000 THEN %MF342 := %MF332 * 4.0 + 2000.0; END_IF;
  //   IF %IW1.5 >= 9500 AND %IW1.5 < 10000 THEN %MD402 := REAL_TO_DINT ( %MF342 ); END_IF;

// Rung 127
  LD [ %IW1.5 >= 10000 ]
  AND [ %IW1.5 < 10500 ]
  [ %MW5 := 13 ]
  [ %MW25 := %IW1.5 - 10000 ]
  [ %MF332 := INT_TO_REAL ( %MW25 ) ]
  [ %MF342 := %MF332 * 8.0 + 4000.0 ]
  [ %MD402 := REAL_TO_DINT ( %MF342 ) ]
  // as ST:
  //   IF %IW1.5 >= 10000 AND %IW1.5 < 10500 THEN %MW5 := 13; END_IF;
  //   IF %IW1.5 >= 10000 AND %IW1.5 < 10500 THEN %MW25 := %IW1.5 - 10000; END_IF;
  //   IF %IW1.5 >= 10000 AND %IW1.5 < 10500 THEN %MF332 := INT_TO_REAL ( %MW25 ); END_IF;
  //   IF %IW1.5 >= 10000 AND %IW1.5 < 10500 THEN %MF342 := %MF332 * 8.0 + 4000.0; END_IF;
  //   IF %IW1.5 >= 10000 AND %IW1.5 < 10500 THEN %MD402 := REAL_TO_DINT ( %MF342 ); END_IF;

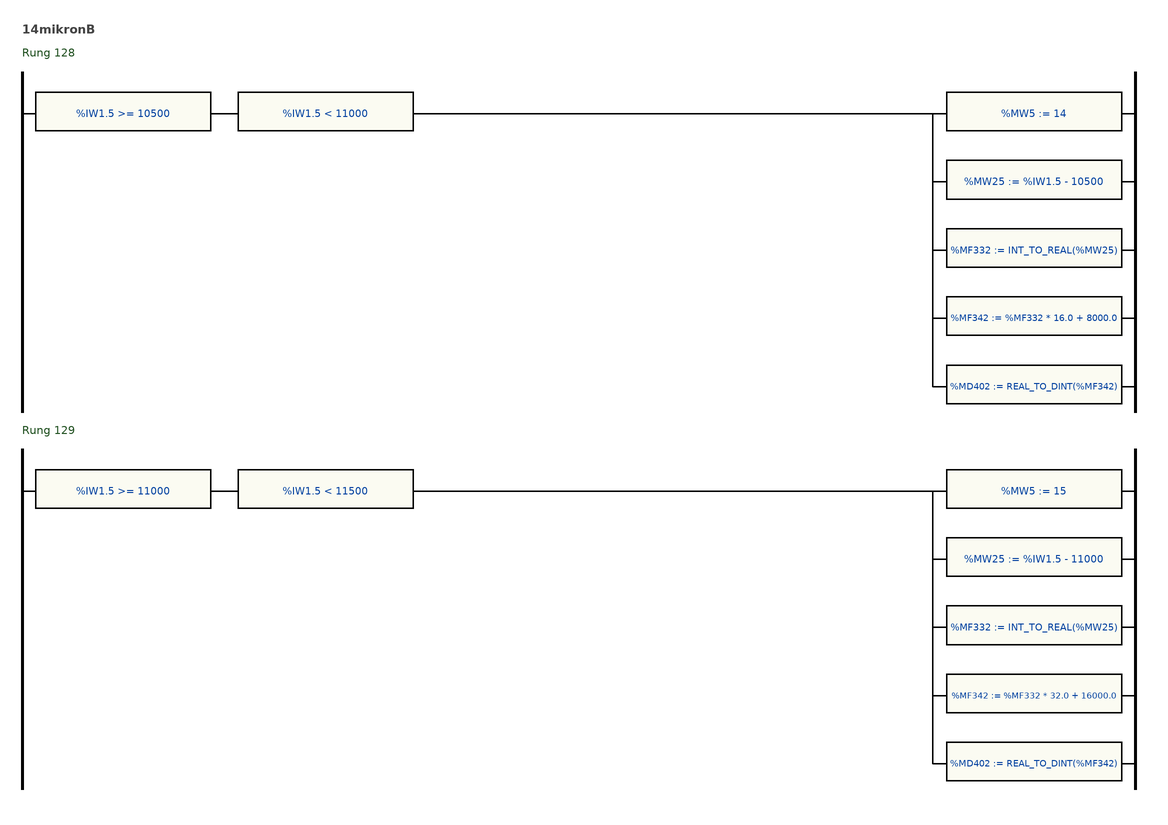

// Rung 128
  LD [ %IW1.5 >= 10500 ]
  AND [ %IW1.5 < 11000 ]
  [ %MW5 := 14 ]
  [ %MW25 := %IW1.5 - 10500 ]
  [ %MF332 := INT_TO_REAL ( %MW25 ) ]
  [ %MF342 := %MF332 * 16.0 + 8000.0 ]
  [ %MD402 := REAL_TO_DINT ( %MF342 ) ]
  // as ST:
  //   IF %IW1.5 >= 10500 AND %IW1.5 < 11000 THEN %MW5 := 14; END_IF;
  //   IF %IW1.5 >= 10500 AND %IW1.5 < 11000 THEN %MW25 := %IW1.5 - 10500; END_IF;
  //   IF %IW1.5 >= 10500 AND %IW1.5 < 11000 THEN %MF332 := INT_TO_REAL ( %MW25 ); END_IF;
  //   IF %IW1.5 >= 10500 AND %IW1.5 < 11000 THEN %MF342 := %MF332 * 16.0 + 8000.0; END_IF;
  //   IF %IW1.5 >= 10500 AND %IW1.5 < 11000 THEN %MD402 := REAL_TO_DINT ( %MF342 ); END_IF;

// Rung 129
  LD [ %IW1.5 >= 11000 ]
  AND [ %IW1.5 < 11500 ]
  [ %MW5 := 15 ]
  [ %MW25 := %IW1.5 - 11000 ]
  [ %MF332 := INT_TO_REAL ( %MW25 ) ]
  [ %MF342 := %MF332 * 32.0 + 16000.0 ]
  [ %MD402 := REAL_TO_DINT ( %MF342 ) ]
  // as ST:
  //   IF %IW1.5 >= 11000 AND %IW1.5 < 11500 THEN %MW5 := 15; END_IF;
  //   IF %IW1.5 >= 11000 AND %IW1.5 < 11500 THEN %MW25 := %IW1.5 - 11000; END_IF;
  //   IF %IW1.5 >= 11000 AND %IW1.5 < 11500 THEN %MF332 := INT_TO_REAL ( %MW25 ); END_IF;
  //   IF %IW1.5 >= 11000 AND %IW1.5 < 11500 THEN %MF342 := %MF332 * 32.0 + 16000.0; END_IF;
  //   IF %IW1.5 >= 11000 AND %IW1.5 < 11500 THEN %MD402 := REAL_TO_DINT ( %MF342 ); END_IF;

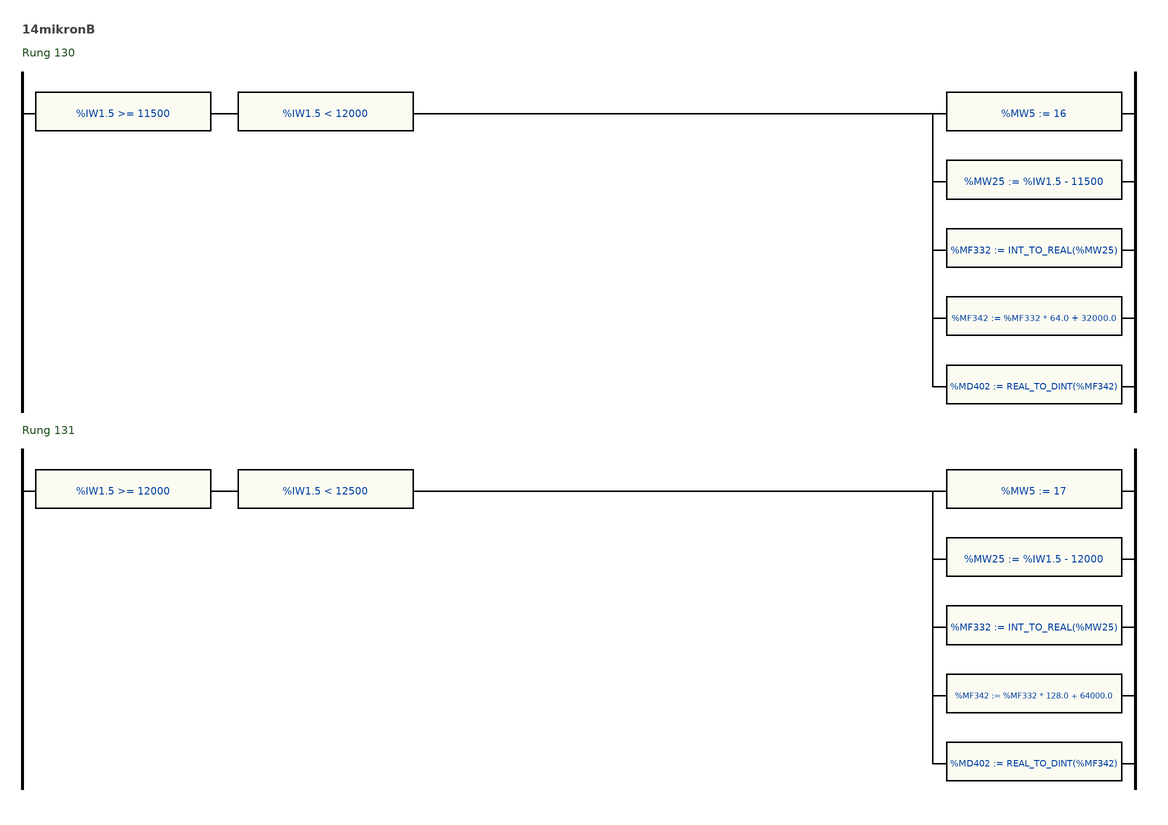

// Rung 130
  LD [ %IW1.5 >= 11500 ]
  AND [ %IW1.5 < 12000 ]
  [ %MW5 := 16 ]
  [ %MW25 := %IW1.5 - 11500 ]
  [ %MF332 := INT_TO_REAL ( %MW25 ) ]
  [ %MF342 := %MF332 * 64.0 + 32000.0 ]
  [ %MD402 := REAL_TO_DINT ( %MF342 ) ]
  // as ST:
  //   IF %IW1.5 >= 11500 AND %IW1.5 < 12000 THEN %MW5 := 16; END_IF;
  //   IF %IW1.5 >= 11500 AND %IW1.5 < 12000 THEN %MW25 := %IW1.5 - 11500; END_IF;
  //   IF %IW1.5 >= 11500 AND %IW1.5 < 12000 THEN %MF332 := INT_TO_REAL ( %MW25 ); END_IF;
  //   IF %IW1.5 >= 11500 AND %IW1.5 < 12000 THEN %MF342 := %MF332 * 64.0 + 32000.0; END_IF;
  //   IF %IW1.5 >= 11500 AND %IW1.5 < 12000 THEN %MD402 := REAL_TO_DINT ( %MF342 ); END_IF;

// Rung 131
  LD [ %IW1.5 >= 12000 ]
  AND [ %IW1.5 < 12500 ]
  [ %MW5 := 17 ]
  [ %MW25 := %IW1.5 - 12000 ]
  [ %MF332 := INT_TO_REAL ( %MW25 ) ]
  [ %MF342 := %MF332 * 128.0 + 64000.0 ]
  [ %MD402 := REAL_TO_DINT ( %MF342 ) ]
  // as ST:
  //   IF %IW1.5 >= 12000 AND %IW1.5 < 12500 THEN %MW5 := 17; END_IF;
  //   IF %IW1.5 >= 12000 AND %IW1.5 < 12500 THEN %MW25 := %IW1.5 - 12000; END_IF;
  //   IF %IW1.5 >= 12000 AND %IW1.5 < 12500 THEN %MF332 := INT_TO_REAL ( %MW25 ); END_IF;
  //   IF %IW1.5 >= 12000 AND %IW1.5 < 12500 THEN %MF342 := %MF332 * 128.0 + 64000.0; END_IF;
  //   IF %IW1.5 >= 12000 AND %IW1.5 < 12500 THEN %MD402 := REAL_TO_DINT ( %MF342 ); END_IF;

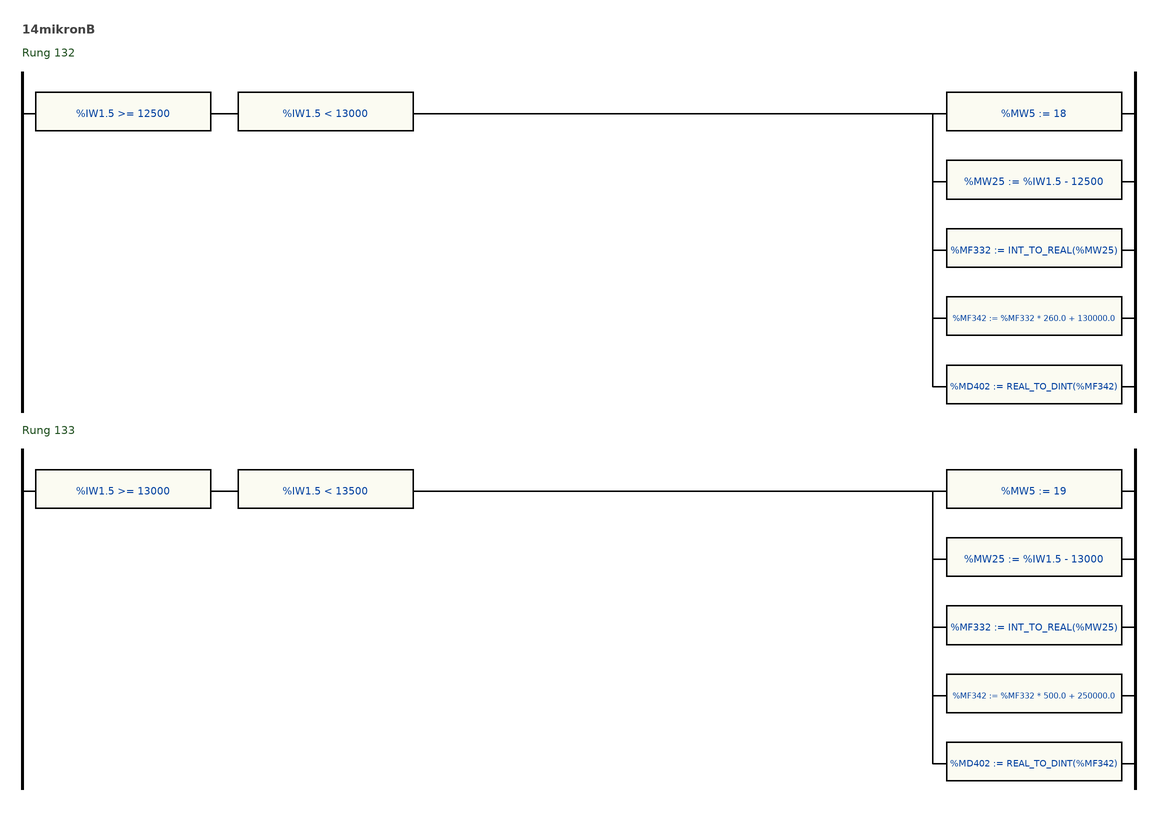

// Rung 132
  LD [ %IW1.5 >= 12500 ]
  AND [ %IW1.5 < 13000 ]
  [ %MW5 := 18 ]
  [ %MW25 := %IW1.5 - 12500 ]
  [ %MF332 := INT_TO_REAL ( %MW25 ) ]
  [ %MF342 := %MF332 * 260.0 + 130000.0 ]
  [ %MD402 := REAL_TO_DINT ( %MF342 ) ]
  // as ST:
  //   IF %IW1.5 >= 12500 AND %IW1.5 < 13000 THEN %MW5 := 18; END_IF;
  //   IF %IW1.5 >= 12500 AND %IW1.5 < 13000 THEN %MW25 := %IW1.5 - 12500; END_IF;
  //   IF %IW1.5 >= 12500 AND %IW1.5 < 13000 THEN %MF332 := INT_TO_REAL ( %MW25 ); END_IF;
  //   IF %IW1.5 >= 12500 AND %IW1.5 < 13000 THEN %MF342 := %MF332 * 260.0 + 130000.0; END_IF;
  //   IF %IW1.5 >= 12500 AND %IW1.5 < 13000 THEN %MD402 := REAL_TO_DINT ( %MF342 ); END_IF;

// Rung 133
  LD [ %IW1.5 >= 13000 ]
  AND [ %IW1.5 < 13500 ]
  [ %MW5 := 19 ]
  [ %MW25 := %IW1.5 - 13000 ]
  [ %MF332 := INT_TO_REAL ( %MW25 ) ]
  [ %MF342 := %MF332 * 500.0 + 250000.0 ]
  [ %MD402 := REAL_TO_DINT ( %MF342 ) ]
  // as ST:
  //   IF %IW1.5 >= 13000 AND %IW1.5 < 13500 THEN %MW5 := 19; END_IF;
  //   IF %IW1.5 >= 13000 AND %IW1.5 < 13500 THEN %MW25 := %IW1.5 - 13000; END_IF;
  //   IF %IW1.5 >= 13000 AND %IW1.5 < 13500 THEN %MF332 := INT_TO_REAL ( %MW25 ); END_IF;
  //   IF %IW1.5 >= 13000 AND %IW1.5 < 13500 THEN %MF342 := %MF332 * 500.0 + 250000.0; END_IF;
  //   IF %IW1.5 >= 13000 AND %IW1.5 < 13500 THEN %MD402 := REAL_TO_DINT ( %MF342 ); END_IF;

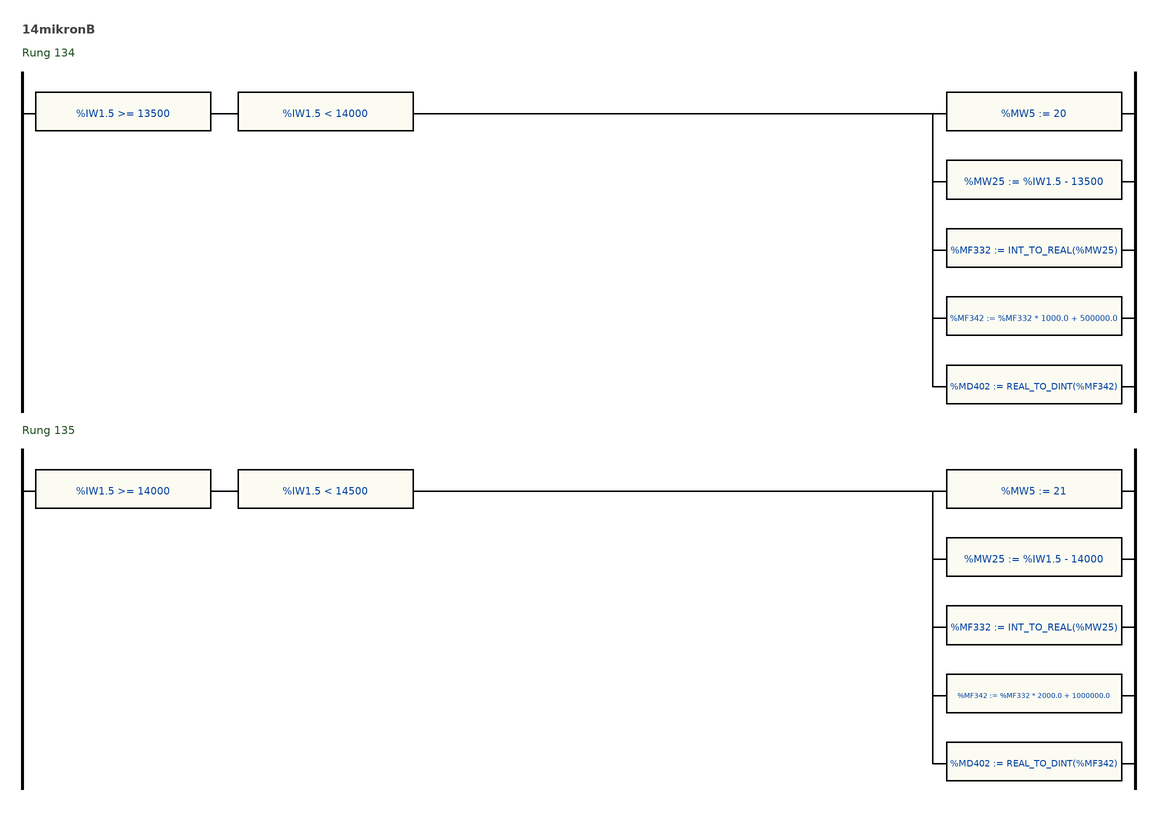

// Rung 134
  LD [ %IW1.5 >= 13500 ]
  AND [ %IW1.5 < 14000 ]
  [ %MW5 := 20 ]
  [ %MW25 := %IW1.5 - 13500 ]
  [ %MF332 := INT_TO_REAL ( %MW25 ) ]
  [ %MF342 := %MF332 * 1000.0 + 500000.0 ]
  [ %MD402 := REAL_TO_DINT ( %MF342 ) ]
  // as ST:
  //   IF %IW1.5 >= 13500 AND %IW1.5 < 14000 THEN %MW5 := 20; END_IF;
  //   IF %IW1.5 >= 13500 AND %IW1.5 < 14000 THEN %MW25 := %IW1.5 - 13500; END_IF;
  //   IF %IW1.5 >= 13500 AND %IW1.5 < 14000 THEN %MF332 := INT_TO_REAL ( %MW25 ); END_IF;
  //   IF %IW1.5 >= 13500 AND %IW1.5 < 14000 THEN %MF342 := %MF332 * 1000.0 + 500000.0; END_IF;
  //   IF %IW1.5 >= 13500 AND %IW1.5 < 14000 THEN %MD402 := REAL_TO_DINT ( %MF342 ); END_IF;

// Rung 135
  LD [ %IW1.5 >= 14000 ]
  AND [ %IW1.5 < 14500 ]
  [ %MW5 := 21 ]
  [ %MW25 := %IW1.5 - 14000 ]
  [ %MF332 := INT_TO_REAL ( %MW25 ) ]
  [ %MF342 := %MF332 * 2000.0 + 1000000.0 ]
  [ %MD402 := REAL_TO_DINT ( %MF342 ) ]
  // as ST:
  //   IF %IW1.5 >= 14000 AND %IW1.5 < 14500 THEN %MW5 := 21; END_IF;
  //   IF %IW1.5 >= 14000 AND %IW1.5 < 14500 THEN %MW25 := %IW1.5 - 14000; END_IF;
  //   IF %IW1.5 >= 14000 AND %IW1.5 < 14500 THEN %MF332 := INT_TO_REAL ( %MW25 ); END_IF;
  //   IF %IW1.5 >= 14000 AND %IW1.5 < 14500 THEN %MF342 := %MF332 * 2000.0 + 1000000.0; END_IF;
  //   IF %IW1.5 >= 14000 AND %IW1.5 < 14500 THEN %MD402 := REAL_TO_DINT ( %MF342 ); END_IF;

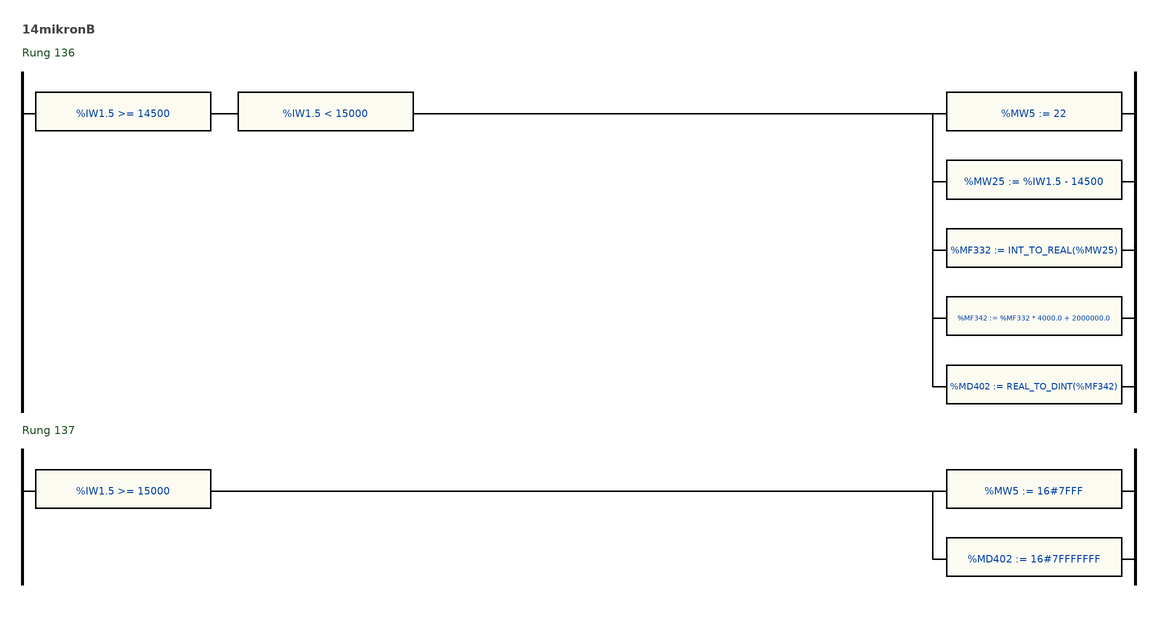

// Rung 136
  LD [ %IW1.5 >= 14500 ]
  AND [ %IW1.5 < 15000 ]
  [ %MW5 := 22 ]
  [ %MW25 := %IW1.5 - 14500 ]
  [ %MF332 := INT_TO_REAL ( %MW25 ) ]
  [ %MF342 := %MF332 * 4000.0 + 2000000.0 ]
  [ %MD402 := REAL_TO_DINT ( %MF342 ) ]
  // as ST:
  //   IF %IW1.5 >= 14500 AND %IW1.5 < 15000 THEN %MW5 := 22; END_IF;
  //   IF %IW1.5 >= 14500 AND %IW1.5 < 15000 THEN %MW25 := %IW1.5 - 14500; END_IF;
  //   IF %IW1.5 >= 14500 AND %IW1.5 < 15000 THEN %MF332 := INT_TO_REAL ( %MW25 ); END_IF;
  //   IF %IW1.5 >= 14500 AND %IW1.5 < 15000 THEN %MF342 := %MF332 * 4000.0 + 2000000.0; END_IF;
  //   IF %IW1.5 >= 14500 AND %IW1.5 < 15000 THEN %MD402 := REAL_TO_DINT ( %MF342 ); END_IF;

// Rung 137
  LD [ %IW1.5 >= 15000 ]
  [ %MW5 := 16#7FFF ]
  [ %MD402 := 16#7FFFFFFF ]
  // as ST:
  //   IF %IW1.5 >= 15000 THEN %MW5 := 16#7FFF; END_IF;
  //   IF %IW1.5 >= 15000 THEN %MD402 := 16#7FFFFFFF; END_IF;

POU DP 1
  (* SectionNumber=7 *)

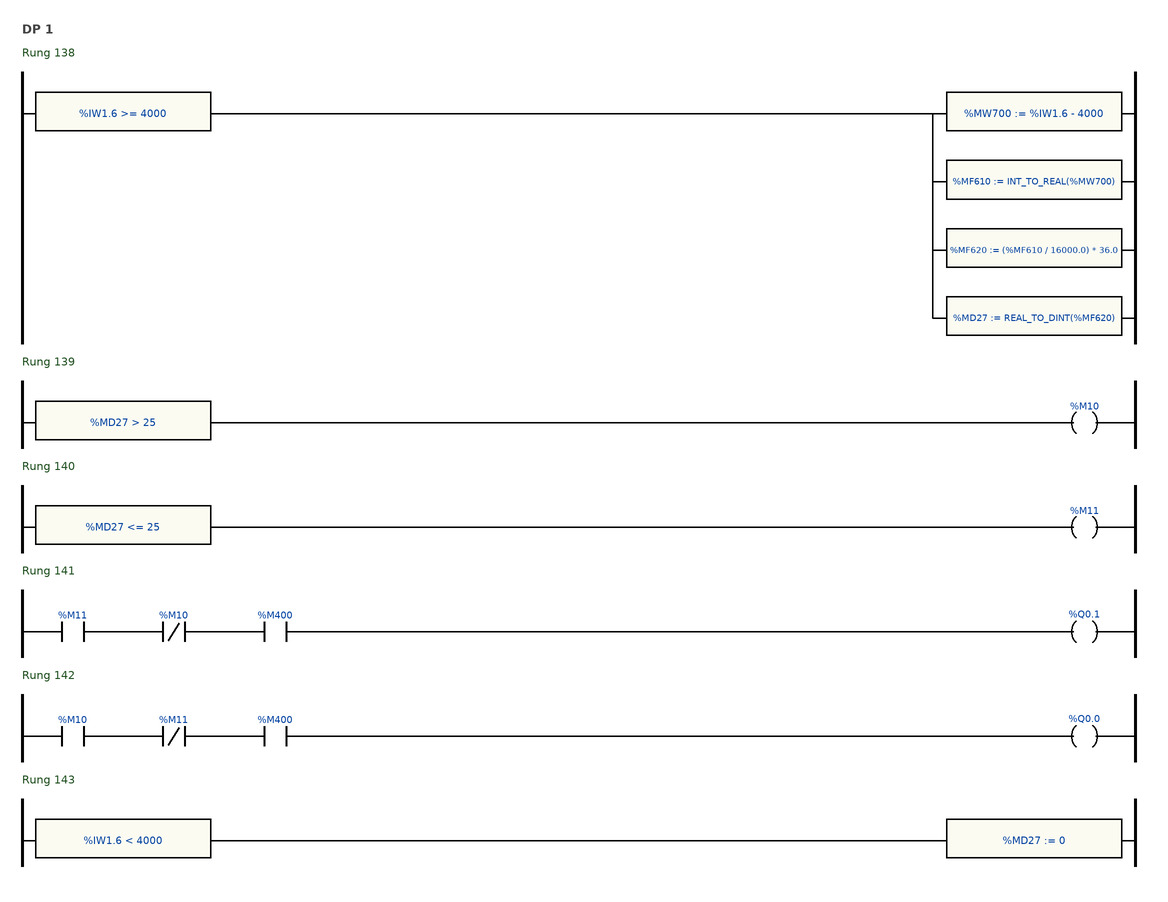

// Rung 138
  LD [ %IW1.6 >= 4000 ]
  [ %MW700 := %IW1.6 - 4000 ]
  [ %MF610 := INT_TO_REAL ( %MW700 ) ]
  [ %MF620 := ( %MF610 / 16000.0 ) * 36.0 ]
  [ %MD27 := REAL_TO_DINT ( %MF620 ) ]
  // as ST:
  //   IF %IW1.6 >= 4000 THEN %MW700 := %IW1.6 - 4000; END_IF;
  //   IF %IW1.6 >= 4000 THEN %MF610 := INT_TO_REAL ( %MW700 ); END_IF;
  //   IF %IW1.6 >= 4000 THEN %MF620 := ( %MF610 / 16000.0 ) * 36.0; END_IF;
  //   IF %IW1.6 >= 4000 THEN %MD27 := REAL_TO_DINT ( %MF620 ); END_IF;

// Rung 139
  LD [ %MD27 > 25 ]
  ST %M10
  // as ST:
  //   %M10 := %MD27 > 25;

// Rung 140
  LD [ %MD27 <= 25 ]
  ST %M11
  // as ST:
  //   %M11 := %MD27 <= 25;

// Rung 141
  LD %M11
  ANDN %M10
  AND %M400
  ST %Q0.1
  // as ST:
  //   %Q0.1 := %M11 AND NOT %M10 AND %M400;

// Rung 142
  LD %M10
  ANDN %M11
  AND %M400
  ST %Q0.0
  // as ST:
  //   %Q0.0 := %M10 AND NOT %M11 AND %M400;

// Rung 143
  LD [ %IW1.6 < 4000 ]
  [ %MD27 := 0 ]
  // as ST:
  //   IF %IW1.6 < 4000 THEN %MD27 := 0; END_IF;

POU DP 2
  (* SectionNumber=8 *)

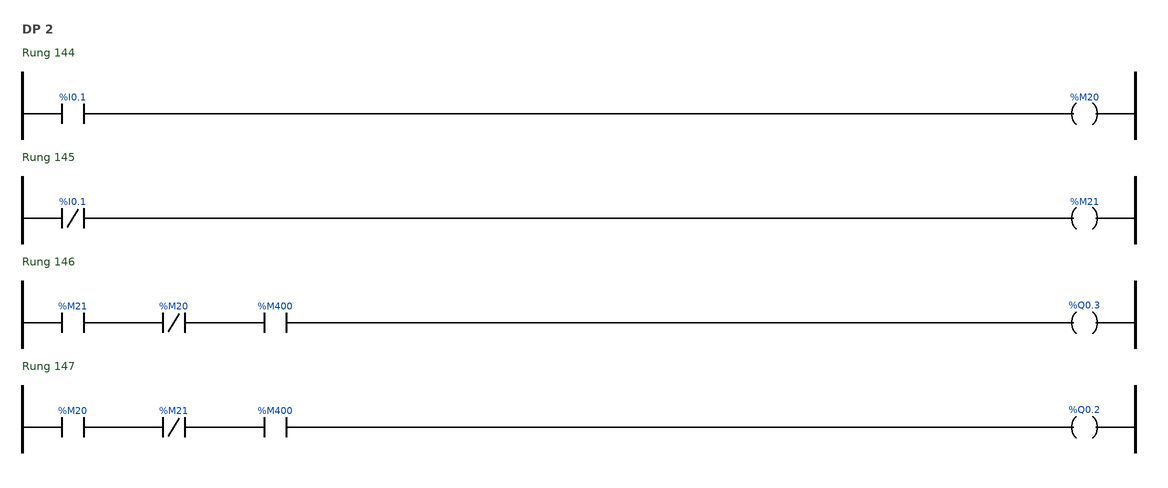

// Rung 144
  LD %I0.1
  ST %M20
  // as ST:
  //   %M20 := %I0.1;

// Rung 145
  LDN %I0.1
  ST %M21
  // as ST:
  //   %M21 := NOT %I0.1;

// Rung 146
  LD %M21
  ANDN %M20
  AND %M400
  ST %Q0.3
  // as ST:
  //   %Q0.3 := %M21 AND NOT %M20 AND %M400;

// Rung 147
  LD %M20
  ANDN %M21
  AND %M400
  ST %Q0.2
  // as ST:
  //   %Q0.2 := %M20 AND NOT %M21 AND %M400;

POU FlowMeter
  (* SectionNumber=9 *)

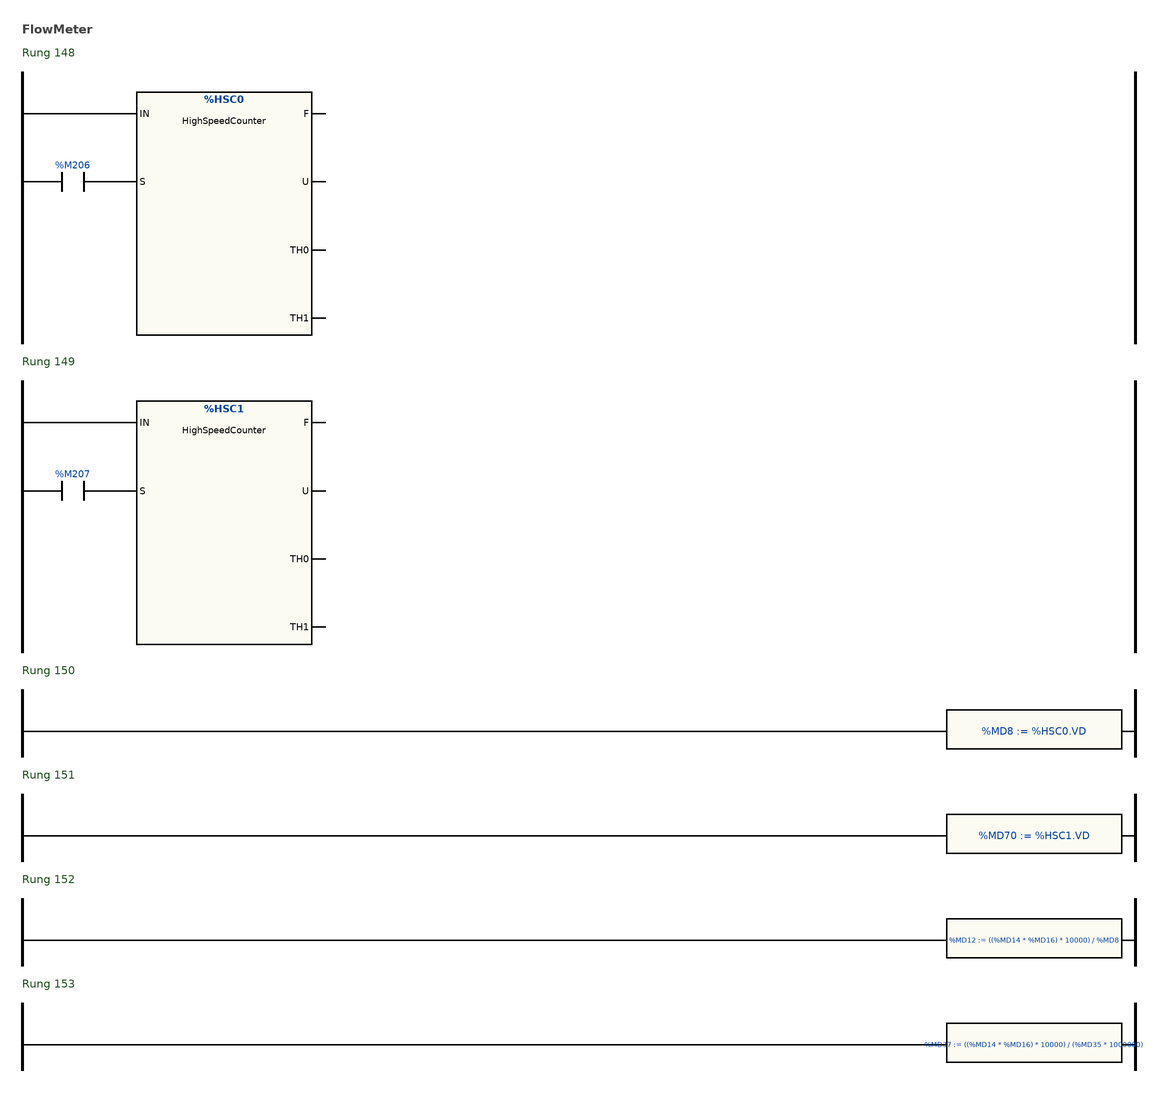

// Rung 148
  BLK %HSC0
  LD 1
  IN
  LD %M206
  S
  END_BLK
  // as ST:
  //   %HSC0(IN := TRUE, S := %M206);

// Rung 149
  BLK %HSC1
  LD 1
  IN
  LD %M207
  S
  END_BLK
  // as ST:
  //   %HSC1(IN := TRUE, S := %M207);

// Rung 150
  LD 1
  [ %MD8 := %HSC0.VD ]
  // as ST:
  //   %MD8 := %HSC0.VD;

// Rung 151
  LD 1
  [ %MD70 := %HSC1.VD ]
  // as ST:
  //   %MD70 := %HSC1.VD;

// Rung 152
  LD 1
  [ %MD12 := ( ( %MD14 * %MD16 ) * 10000 ) / %MD8 ]
  // as ST:
  //   %MD12 := ( ( %MD14 * %MD16 ) * 10000 ) / %MD8;

// Rung 153
  LD 1
  [ %MD37 := ( ( %MD14 * %MD16 ) * 10000 ) / ( %MD35 * 1000000 ) ]
  // as ST:
  //   %MD37 := ( ( %MD14 * %MD16 ) * 10000 ) / ( %MD35 * 1000000 );

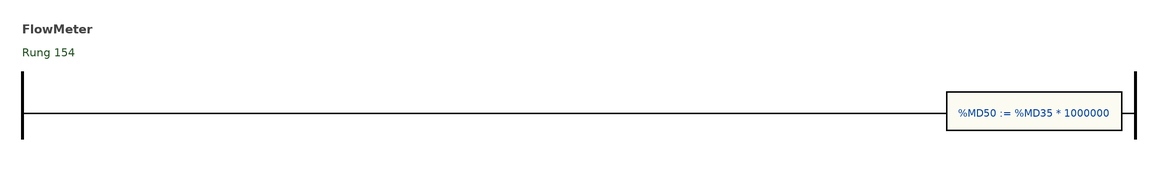

// Rung 154
  LD 1
  [ %MD50 := %MD35 * 1000000 ]
  // as ST:
  //   %MD50 := %MD35 * 1000000;

POU Solenoid
  (* SectionNumber=10 *)

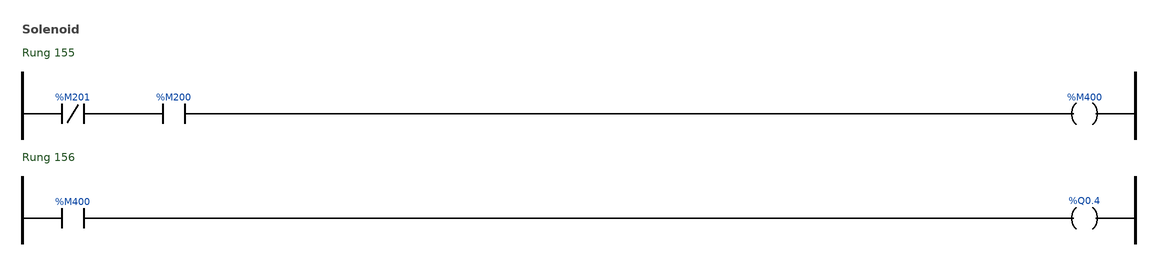

// Rung 155
  LDN %M201
  AND %M200
  ST %M400
  // as ST:
  //   %M400 := NOT %M201 AND %M200;

// Rung 156
  LD %M400
  ST %Q0.4
  // as ST:
  //   %Q0.4 := %M400;

POU Warning
  (* SectionNumber=11 *)

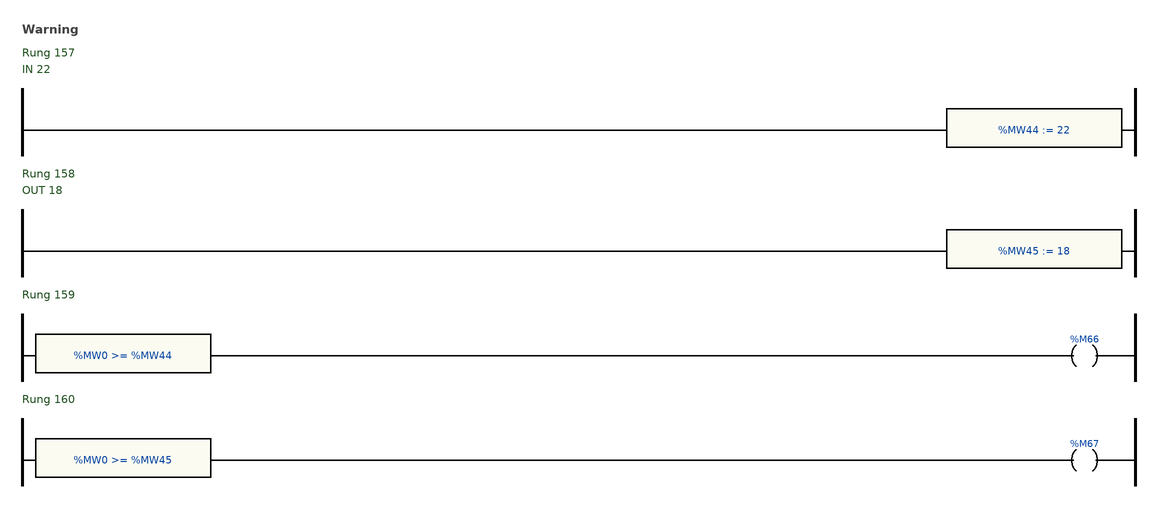

// Rung 157
// IN 22
  LD 1
  [ %MW44 := 22 ]
  // as ST:
  //   %MW44 := 22;

// Rung 158
// OUT 18
  LD 1
  [ %MW45 := 18 ]
  // as ST:
  //   %MW45 := 18;

// Rung 159
  LD [ %MW0 >= %MW44 ]
  ST %M66
  // as ST:
  //   %M66 := %MW0 >= %MW44;

// Rung 160
  LD [ %MW0 >= %MW45 ]
  ST %M67
  // as ST:
  //   %M67 := %MW0 >= %MW45;

POU FilterQuality
  (* SectionNumber=12 *)

